   cmMendrelCathodeFrontAxisZ.commandConfiguration.camIn.deceleration := -1.0;
   cmMendrelCathodeFrontAxisZ.commandConfiguration.camIn.jerk := -1.0;
   cmMendrelCathodeFrontAxisZ.commandConfiguration.camIn.applicationMode := 0;
   cmMendrelCathodeFrontAxisZ.commandConfiguration.camIn.syncDirection := 1;
   cmMendrelCathodeFrontAxisZ.commandConfiguration.gearOutCamOut.slavePosition := 0.0;
   cmMendrelCathodeFrontAxisZ.commandConfiguration.gearOutCamOut.syncProfileReference := 1;
   cmMendrelCathodeFrontAxisZ.commandConfiguration.gearOutCamOut.masterStopDistance := 0.0;
   cmMendrelCathodeFrontAxisZ.commandConfiguration.gearOutCamOut.deceleration := -1.0;
   cmMendrelCathodeFrontAxisZ.commandConfiguration.gearOutCamOut.jerk := -1.0;
   cmMendrelCathodeFrontAxisZ.commandConfiguration.gearOutCamOut.syncOutDirection := 3;
   cmMendrelCathodeFrontAxisZ.commandConfiguration.gearOutCamOut.gearOutCamOutMode := -1;
   cmMendrelCathodeFrontAxisZ.commandConfiguration.phasing.phaseShift := 0.0;
   cmMendrelCathodeFrontAxisZ.commandConfiguration.phasing.velocity := -1.0;
   cmMendrelCathodeFrontAxisZ.commandConfiguration.phasing.acceleration := -1.0;
   cmMendrelCathodeFrontAxisZ.commandConfiguration.phasing.deceleration := -1.0;
   cmMendrelCathodeFrontAxisZ.commandConfiguration.phasing.jerk := -1.0;
   cmMendrelCathodeFrontAxisZ.commandConfiguration.phasing.profileReference := 0;
   cmMendrelCathodeFrontAxisZ.commandConfiguration.phasing.phasingDistance := 0.0;
   cmMendrelCathodeFrontAxisZ.commandConfiguration.phasing.startPosition := 0.0;
   cmMendrelCathodeFrontAxisZ.commandConfiguration.phasing.direction := 3;
   cmMendrelCathodeFrontAxisZ.commandConfiguration.phasing.phaseAbsolute := TRUE;
   cmMendrelCathodeFrontAxisZ.commandConfiguration.phasing.phaseShiftChangeOnTheFly := FALSE;
   cmMendrelCathodeFrontAxisZ.commandConfiguration.offset.offset := 0.0;
   cmMendrelCathodeFrontAxisZ.commandConfiguration.offset.profileReference := 1;
   cmMendrelCathodeFrontAxisZ.commandConfiguration.offset.offsetDistance := 0.0;
   cmMendrelCathodeFrontAxisZ.commandConfiguration.offset.startPosition := 0.0;
   cmMendrelCathodeFrontAxisZ.commandConfiguration.offset.direction := 3;
   cmMendrelCathodeFrontAxisZ.commandConfiguration.offset.offsetAbsolute := TRUE;
   cmMendrelCathodeFrontAxisZ.commandConfiguration.offset.offsetChangeOnTheFly := FALSE;
   cmMendrelCathodeFrontAxisZ.commands.enableMasterControl := TRUE;
   cmMendrelCathodeFrontAxisZ.commands.enableAxis := FALSE;
   cmMendrelCathodeFrontAxisZ.commands.resetAxis := FALSE;
   cmMendrelCathodeFrontAxisZ.commands.openBrake := FALSE;
   cmMendrelCathodeFrontAxisZ.commands.jogForward := FALSE;
   cmMendrelCathodeFrontAxisZ.commands.jogBackward := FALSE;
   cmMendrelCathodeFrontAxisZ.commands.moveVelocity := FALSE;
   cmMendrelCathodeFrontAxisZ.commands.stop := FALSE;
   cmMendrelCathodeFrontAxisZ.commands.fastStop := FALSE;
   cmMendrelCathodeFrontAxisZ.commands.torqueLimiting := FALSE;
   cmMendrelCathodeFrontAxisZ.commands.homing := FALSE;
   cmMendrelCathodeFrontAxisZ.commands.posRelative := FALSE;
   cmMendrelCathodeFrontAxisZ.commands.posAbsolute := FALSE;
   cmMendrelCathodeFrontAxisZ.commands.posSuperimposed := FALSE;
   cmMendrelCathodeFrontAxisZ.commands.haltSuperimposed := FALSE;
   cmMendrelCathodeFrontAxisZ.commands.selectSetPosition := 1;
   cmMendrelCathodeFrontAxisZ.commands.uploadParameters := FALSE;
   cmMendrelCathodeFrontAxisZ.commands.refreshConfiguration := FALSE;
   cmMendrelCathodeFrontAxisZ.commands.editConfiguration := FALSE;
   cmMendrelCathodeFrontAxisZ.commands.saveConfiguration := FALSE;
   cmMendrelCathodeFrontAxisZ.commands.uploadCurrentTorque := FALSE;
   cmMendrelCathodeFrontAxisZ.commands.reset := FALSE;
   cmMendrelCathodeFrontAxisZ.monitoring.enable := TRUE;
   cmMendrelCathodeFrontAxisZ.monitoring.referenceDesignator := WSTRING#'MendrelCathodeFrontAxisZ';
   cmMendrelCathodeFrontAxisZ.monitoring.enabled := TRUE;
   cmMendrelCathodeFrontAxisZ.monitoring.enableManualCmds := FALSE;
   cmMendrelCathodeFrontAxisZ.monitoring.reset := FALSE;
   cmMendrelCathodeFrontAxisZ.monitoring.resetAxis := FALSE;
   cmMendrelCathodeFrontAxisZ.monitoring.enableAxis := TRUE;
   cmMendrelCathodeFrontAxisZ.monitoring.openBrake := FALSE;
   cmMendrelCathodeFrontAxisZ.monitoring.jogBackward := FALSE;
   cmMendrelCathodeFrontAxisZ.monitoring.jogForward := FALSE;
   cmMendrelCathodeFrontAxisZ.monitoring.moveVelocity := FALSE;
   cmMendrelCathodeFrontAxisZ.monitoring.stop := FALSE;
   cmMendrelCathodeFrontAxisZ.monitoring.fastStop := FALSE;
   cmMendrelCathodeFrontAxisZ.monitoring.torqueLimiting := FALSE;
   cmMendrelCathodeFrontAxisZ.monitoring.homing := FALSE;
   cmMendrelCathodeFrontAxisZ.monitoring.posRelative := FALSE;
   cmMendrelCathodeFrontAxisZ.monitoring.posAbsolute := FALSE;
   cmMendrelCathodeFrontAxisZ.monitoring.posSuperimposed := FALSE;
   cmMendrelCathodeFrontAxisZ.monitoring.haltSuperimposed := FALSE;
   cmMendrelCathodeFrontAxisZ.monitoring.brakeOpened := FALSE;
   cmMendrelCathodeFrontAxisZ.monitoring.axisEnabled := TRUE;
   cmMendrelCathodeFrontAxisZ.monitoring.resetActive := FALSE;
   cmMendrelCathodeFrontAxisZ.monitoring.inVelocity := FALSE;
   cmMendrelCathodeFrontAxisZ.monitoring.inLimitation := FALSE;
   cmMendrelCathodeFrontAxisZ.monitoring.inClamping := FALSE;
   cmMendrelCathodeFrontAxisZ.monitoring.startSync := FALSE;
   cmMendrelCathodeFrontAxisZ.monitoring.inSync := FALSE;
   cmMendrelCathodeFrontAxisZ.monitoring.inSimulation := FALSE;
   cmMendrelCathodeFrontAxisZ.monitoring.jogSelected := FALSE;
   cmMendrelCathodeFrontAxisZ.monitoring.moveVelocitySelected := FALSE;
   cmMendrelCathodeFrontAxisZ.monitoring.stopSelected := FALSE;
   cmMendrelCathodeFrontAxisZ.monitoring.fastStopSelected := FALSE;
   cmMendrelCathodeFrontAxisZ.monitoring.torqueLimitingSelected := FALSE;
   cmMendrelCathodeFrontAxisZ.monitoring.homingSelected := FALSE;
   cmMendrelCathodeFrontAxisZ.monitoring.posRelativeSelected := FALSE;
   cmMendrelCathodeFrontAxisZ.monitoring.posAbsoluteSelected := FALSE;
   cmMendrelCathodeFrontAxisZ.monitoring.posSuperimposedSelected := FALSE;
   cmMendrelCathodeFrontAxisZ.monitoring.haltSuperimposedSelected := FALSE;
   cmMendrelCathodeFrontAxisZ.monitoring.commandBusy := FALSE;
   cmMendrelCathodeFrontAxisZ.monitoring.commandDone := FALSE;
   cmMendrelCathodeFrontAxisZ.monitoring.commandAborted := FALSE;
   cmMendrelCathodeFrontAxisZ.monitoring.homingCommandBusy := FALSE;
   cmMendrelCathodeFrontAxisZ.monitoring.homingCommandDone := FALSE;
   cmMendrelCathodeFrontAxisZ.monitoring.homingCommandAborted := FALSE;
   cmMendrelCathodeFrontAxisZ.monitoring.superimposedBusy := FALSE;
   cmMendrelCathodeFrontAxisZ.monitoring.superimposedDone := FALSE;
   cmMendrelCathodeFrontAxisZ.monitoring.superimposedAborted := FALSE;
   cmMendrelCathodeFrontAxisZ.monitoring.selectSetPosition := 1;
   cmMendrelCathodeFrontAxisZ.monitoring.selectionController := FALSE;
   cmMendrelCathodeFrontAxisZ.monitoring.interlockGeneral := TRUE;
   cmMendrelCathodeFrontAxisZ.monitoring.interlockJogForward := TRUE;
   cmMendrelCathodeFrontAxisZ.monitoring.interlockJogBackward := TRUE;
   cmMendrelCathodeFrontAxisZ.monitoring.interlockWarningGeneral := FALSE;
   cmMendrelCathodeFrontAxisZ.monitoring.interlockWarningJogForward := FALSE;
   cmMendrelCathodeFrontAxisZ.monitoring.interlockWarningJogBackward := FALSE;
   cmMendrelCathodeFrontAxisZ.monitoring.valid := TRUE;
   cmMendrelCathodeFrontAxisZ.monitoring.busy := TRUE;
   cmMendrelCathodeFrontAxisZ.monitoring.error := FALSE;
   cmMendrelCathodeFrontAxisZ.monitoring.status := 16#7002;
   cmMendrelCathodeFrontAxisZ.monitoring.subfunctionStatus := 16#0000;
   cmMendrelCathodeFrontAxisZ.monitoring.actualPosition := 50.0;
   cmMendrelCathodeFrontAxisZ.monitoring.actualSpeed := 0.0;
   cmMendrelCathodeFrontAxisZ.monitoring.speedUnit := 1062;
   cmMendrelCathodeFrontAxisZ.monitoring.positionUnit := 1013;
   cmMendrelCathodeFrontAxisZ.monitoring.axisStatus1 := 16#0240_10A1;
   cmMendrelCathodeFrontAxisZ.monitoring.axisStatus2 := 16#0000_0000;
   cmMendrelCathodeFrontAxisZ.monitoring.axisType := 1;
   cmMendrelCathodeFrontAxisZ.monitoring.maxVelocity := 2500.0;
   cmMendrelCathodeFrontAxisZ.monitoring.actualCurrent := 0.0;
   cmMendrelCathodeFrontAxisZ.monitoring.actualTorque := 0.0;
   cmMendrelCathodeFrontAxisZ.monitoring.velocityOverrideEnabled := FALSE;
   cmMendrelCathodeFrontAxisZ.monitoring.sinaParaError := FALSE;
   cmMendrelCathodeFrontAxisZ.monitoring.sinaParaStatus := 16#0000_0000;
   cmMendrelCathodeFrontAxisZ.configuration.referenceDesignator := WSTRING#'MendrelCathodeFrontAxisZ';
   cmMendrelCathodeFrontAxisZ.configuration.disableAlarms := FALSE;
   cmMendrelCathodeFrontAxisZ.configuration.masterControlPopUp := TRUE;
   cmMendrelCathodeFrontAxisZ.configuration.setPositions[0].position := 0.0;
   cmMendrelCathodeFrontAxisZ.configuration.setPositions[1].position := 50.0;
   cmMendrelCathodeFrontAxisZ.configuration.setPositions[2..15].position := 0.0;
   cmMendrelCathodeFrontAxisZ.configuration.setPositions[0..1].velocity := 50.0;
   cmMendrelCathodeFrontAxisZ.configuration.setPositions[2..15].velocity := -1.0;
   cmMendrelCathodeFrontAxisZ.configuration.setPositions[0..1].acceleration := 500.0;
   cmMendrelCathodeFrontAxisZ.configuration.setPositions[2..15].acceleration := -1.0;
   cmMendrelCathodeFrontAxisZ.configuration.setPositions[0..1].deceleration := 500.0;
   cmMendrelCathodeFrontAxisZ.configuration.setPositions[2..15].deceleration := -1.0;
   cmMendrelCathodeFrontAxisZ.configuration.setPositions[0..15]."name" := '';
   cmMendrelCathodeRearAxisY.commandConfiguration.generalSettings.stopOnError := TRUE;
   cmMendrelCathodeRearAxisY.commandConfiguration.generalSettings.resetWithRestart := FALSE;
   cmMendrelCathodeRearAxisY.commandConfiguration.generalSettings.abortWaitingSyncCmd := TRUE;
   cmMendrelCathodeRearAxisY.commandConfiguration.power.startMode := 1;
   cmMendrelCathodeRearAxisY.commandConfiguration.power.stopMode := 0;
   cmMendrelCathodeRearAxisY.commandConfiguration.power.syncMotionSimulation := FALSE;
   cmMendrelCathodeRearAxisY.commandConfiguration.power.syncMotionSimulationExtendedMode := -1;
   cmMendrelCathodeRearAxisY.commandConfiguration.jog.velocity := 0.0;
   cmMendrelCathodeRearAxisY.commandConfiguration.jog.acceleration := -1.0;
   cmMendrelCathodeRearAxisY.commandConfiguration.jog.deceleration := -1.0;
   cmMendrelCathodeRearAxisY.commandConfiguration.jog.jerk := -1.0;
   cmMendrelCathodeRearAxisY.commandConfiguration.jog.positionControlled := TRUE;
   cmMendrelCathodeRearAxisY.commandConfiguration.jog.increment := 0.0;
   cmMendrelCathodeRearAxisY.commandConfiguration.jog.mode := 0;
   cmMendrelCathodeRearAxisY.commandConfiguration.moveVelocity.velocity := 0.0;
   cmMendrelCathodeRearAxisY.commandConfiguration.moveVelocity.acceleration := -1.0;
   cmMendrelCathodeRearAxisY.commandConfiguration.moveVelocity.deceleration := -1.0;
   cmMendrelCathodeRearAxisY.commandConfiguration.moveVelocity.jerk := -1.0;
   cmMendrelCathodeRearAxisY.commandConfiguration.moveVelocity.direction := 0;
   cmMendrelCathodeRearAxisY.commandConfiguration.moveVelocity.positionControlled := TRUE;
   cmMendrelCathodeRearAxisY.commandConfiguration.moveVelocity.velocityChangeOnTheFly := FALSE;
   cmMendrelCathodeRearAxisY.commandConfiguration.stop.deceleration := -1.0;
   cmMendrelCathodeRearAxisY.commandConfiguration.stop.jerk := -1.0;
   cmMendrelCathodeRearAxisY.commandConfiguration.stop.abortAcceleration := FALSE;
   cmMendrelCathodeRearAxisY.commandConfiguration.fastStop.deceleration := -1.0;
   cmMendrelCathodeRearAxisY.commandConfiguration.fastStop.jerk := -1.0;
   cmMendrelCathodeRearAxisY.commandConfiguration.fastStop.abortAcceleration := FALSE;
   cmMendrelCathodeRearAxisY.commandConfiguration.fastStop.replaceStopPossible := FALSE;
   cmMendrelCathodeRearAxisY.commandConfiguration.torqueLimiting.limit := -1.0;
   cmMendrelCathodeRearAxisY.commandConfiguration.torqueLimiting.mode := 0;
   cmMendrelCathodeRearAxisY.commandConfiguration.homing.position := 0.0;
   cmMendrelCathodeRearAxisY.commandConfiguration.homing.mode := 0;
   cmMendrelCathodeRearAxisY.commandConfiguration.homing.sensor := 0;
   cmMendrelCathodeRearAxisY.commandConfiguration.homing.extendedMode := -1;
   cmMendrelCathodeRearAxisY.commandConfiguration.homing.extendedModeTorqueLimit := 0.0;
   cmMendrelCathodeRearAxisY.commandConfiguration.homing.extendedModeTargetPosition := 0.0;
   cmMendrelCathodeRearAxisY.commandConfiguration.posRelative.distance := 0.0;
   cmMendrelCathodeRearAxisY.commandConfiguration.posRelative.velocity := -1.0;
   cmMendrelCathodeRearAxisY.commandConfiguration.posRelative.acceleration := -1.0;
   cmMendrelCathodeRearAxisY.commandConfiguration.posRelative.deceleration := -1.0;
   cmMendrelCathodeRearAxisY.commandConfiguration.posRelative.jerk := -1.0;
   cmMendrelCathodeRearAxisY.commandConfiguration.posRelative.direction := 0;
   cmMendrelCathodeRearAxisY.commandConfiguration.posAbsolute.position := 0.0;
   cmMendrelCathodeRearAxisY.commandConfiguration.posAbsolute.velocity := -1.0;
   cmMendrelCathodeRearAxisY.commandConfiguration.posAbsolute.acceleration := -1.0;
   cmMendrelCathodeRearAxisY.commandConfiguration.posAbsolute.deceleration := -1.0;
   cmMendrelCathodeRearAxisY.commandConfiguration.posAbsolute.jerk := -1.0;
   cmMendrelCathodeRearAxisY.commandConfiguration.posAbsolute.direction := 1;
   cmMendrelCathodeRearAxisY.commandConfiguration.posAbsolute.positionChangeOnTheFly := FALSE;
   cmMendrelCathodeRearAxisY.commandConfiguration.posAbsolute.velocityChangeOnTheFly := FALSE;
   cmMendrelCathodeRearAxisY.commandConfiguration.posSuperimposed.distance := 0.0;
   cmMendrelCathodeRearAxisY.commandConfiguration.posSuperimposed.velocityDiff := -1.0;
   cmMendrelCathodeRearAxisY.commandConfiguration.posSuperimposed.acceleration := -1.0;
   cmMendrelCathodeRearAxisY.commandConfiguration.posSuperimposed.deceleration := -1.0;
   cmMendrelCathodeRearAxisY.commandConfiguration.posSuperimposed.jerk := -1.0;
   cmMendrelCathodeRearAxisY.commandConfiguration.posSuperimposed.direction := 0;
   cmMendrelCathodeRearAxisY.commandConfiguration.haltSuperimposed.deceleration := -1.0;
   cmMendrelCathodeRearAxisY.commandConfiguration.haltSuperimposed.jerk := -1.0;
   cmMendrelCathodeRearAxisY.commandConfiguration.haltSuperimposed.abortAcceleration := FALSE;
   cmMendrelCathodeRearAxisY.commandConfiguration.gearInRelative.ratioNumerator := 1;
   cmMendrelCathodeRearAxisY.commandConfiguration.gearInRelative.ratioDenominator := 1;
   cmMendrelCathodeRearAxisY.commandConfiguration.gearInRelative.acceleration := -1.0;
   cmMendrelCathodeRearAxisY.commandConfiguration.gearInRelative.deceleration := -1.0;
   cmMendrelCathodeRearAxisY.commandConfiguration.gearInRelative.jerk := -1.0;
   cmMendrelCathodeRearAxisY.commandConfiguration.gearInRelative.ratioChangeOnTheFly := FALSE;
   cmMendrelCathodeRearAxisY.commandConfiguration.gearInAbsolute.ratioNumerator := 1;
   cmMendrelCathodeRearAxisY.commandConfiguration.gearInAbsolute.ratioDenominator := 1;
   cmMendrelCathodeRearAxisY.commandConfiguration.gearInAbsolute.masterSyncPosition := 0.0;
   cmMendrelCathodeRearAxisY.commandConfiguration.gearInAbsolute.slaveSyncPosition := 0.0;
   cmMendrelCathodeRearAxisY.commandConfiguration.gearInAbsolute.syncProfileReference := 1;
   cmMendrelCathodeRearAxisY.commandConfiguration.gearInAbsolute.masterStartDistance := 0.0;
   cmMendrelCathodeRearAxisY.commandConfiguration.gearInAbsolute.velocity := -1.0;
   cmMendrelCathodeRearAxisY.commandConfiguration.gearInAbsolute.acceleration := -1.0;
   cmMendrelCathodeRearAxisY.commandConfiguration.gearInAbsolute.deceleration := -1.0;
   cmMendrelCathodeRearAxisY.commandConfiguration.gearInAbsolute.jerk := -1.0;
   cmMendrelCathodeRearAxisY.commandConfiguration.gearInAbsolute.syncDirection := 1;
   cmMendrelCathodeRearAxisY.commandConfiguration.gearInAbsolute.ratioChangeOnTheFly := FALSE;
   cmMendrelCathodeRearAxisY.commandConfiguration.gearInVelocity.continuousUpdate := FALSE;
   cmMendrelCathodeRearAxisY.commandConfiguration.gearInVelocity.ratioNumerator := 1;
   cmMendrelCathodeRearAxisY.commandConfiguration.gearInVelocity.ratioDenominator := 1;
   cmMendrelCathodeRearAxisY.commandConfiguration.gearInVelocity.acceleration := -1.0;
   cmMendrelCathodeRearAxisY.commandConfiguration.gearInVelocity.deceleration := -1.0;
   cmMendrelCathodeRearAxisY.commandConfiguration.gearInVelocity.jerk := -1.0;
   cmMendrelCathodeRearAxisY.commandConfiguration.gearInVelocity.positionControlled := FALSE;
   cmMendrelCathodeRearAxisY.commandConfiguration.camIn.masterOffset := 0.0;
   cmMendrelCathodeRearAxisY.commandConfiguration.camIn.slaveOffset := 0.0;
   cmMendrelCathodeRearAxisY.commandConfiguration.camIn.masterScaling := 1.0;
   cmMendrelCathodeRearAxisY.commandConfiguration.camIn.slaveScaling := 1.0;
   cmMendrelCathodeRearAxisY.commandConfiguration.camIn.masterSyncPosition := 0.0;
   cmMendrelCathodeRearAxisY.commandConfiguration.camIn.syncProfileReference := 1;
   cmMendrelCathodeRearAxisY.commandConfiguration.camIn.masterStartDistance := 0.0;
   cmMendrelCathodeRearAxisY.commandConfiguration.camIn.velocity := -1.0;
   cmMendrelCathodeRearAxisY.commandConfiguration.camIn.acceleration := -1.0;
   cmMendrelCathodeRearAxisY.commandConfiguration.camIn.deceleration := -1.0;
   cmMendrelCathodeRearAxisY.commandConfiguration.camIn.jerk := -1.0;
   cmMendrelCathodeRearAxisY.commandConfiguration.camIn.applicationMode := 0;
   cmMendrelCathodeRearAxisY.commandConfiguration.camIn.syncDirection := 1;
   cmMendrelCathodeRearAxisY.commandConfiguration.gearOutCamOut.slavePosition := 0.0;
   cmMendrelCathodeRearAxisY.commandConfiguration.gearOutCamOut.syncProfileReference := 1;
   cmMendrelCathodeRearAxisY.commandConfiguration.gearOutCamOut.masterStopDistance := 0.0;
   cmMendrelCathodeRearAxisY.commandConfiguration.gearOutCamOut.deceleration := -1.0;
   cmMendrelCathodeRearAxisY.commandConfiguration.gearOutCamOut.jerk := -1.0;
   cmMendrelCathodeRearAxisY.commandConfiguration.gearOutCamOut.syncOutDirection := 3;
   cmMendrelCathodeRearAxisY.commandConfiguration.gearOutCamOut.gearOutCamOutMode := -1;
   cmMendrelCathodeRearAxisY.commandConfiguration.phasing.phaseShift := 0.0;
   cmMendrelCathodeRearAxisY.commandConfiguration.phasing.velocity := -1.0;
   cmMendrelCathodeRearAxisY.commandConfiguration.phasing.acceleration := -1.0;
   cmMendrelCathodeRearAxisY.commandConfiguration.phasing.deceleration := -1.0;
   cmMendrelCathodeRearAxisY.commandConfiguration.phasing.jerk := -1.0;
   cmMendrelCathodeRearAxisY.commandConfiguration.phasing.profileReference := 0;
   cmMendrelCathodeRearAxisY.commandConfiguration.phasing.phasingDistance := 0.0;
   cmMendrelCathodeRearAxisY.commandConfiguration.phasing.startPosition := 0.0;
   cmMendrelCathodeRearAxisY.commandConfiguration.phasing.direction := 3;
   cmMendrelCathodeRearAxisY.commandConfiguration.phasing.phaseAbsolute := TRUE;
   cmMendrelCathodeRearAxisY.commandConfiguration.phasing.phaseShiftChangeOnTheFly := FALSE;
   cmMendrelCathodeRearAxisY.commandConfiguration.offset.offset := 0.0;
   cmMendrelCathodeRearAxisY.commandConfiguration.offset.profileReference := 1;
   cmMendrelCathodeRearAxisY.commandConfiguration.offset.offsetDistance := 0.0;
   cmMendrelCathodeRearAxisY.commandConfiguration.offset.startPosition := 0.0;
   cmMendrelCathodeRearAxisY.commandConfiguration.offset.direction := 3;
   cmMendrelCathodeRearAxisY.commandConfiguration.offset.offsetAbsolute := TRUE;
   cmMendrelCathodeRearAxisY.commandConfiguration.offset.offsetChangeOnTheFly := FALSE;
   cmMendrelCathodeRearAxisY.commands.enableMasterControl := TRUE;
   cmMendrelCathodeRearAxisY.commands.enableAxis := FALSE;
   cmMendrelCathodeRearAxisY.commands.resetAxis := FALSE;
   cmMendrelCathodeRearAxisY.commands.openBrake := FALSE;
   cmMendrelCathodeRearAxisY.commands.jogForward := FALSE;
   cmMendrelCathodeRearAxisY.commands.jogBackward := FALSE;
   cmMendrelCathodeRearAxisY.commands.moveVelocity := FALSE;
   cmMendrelCathodeRearAxisY.commands.stop := FALSE;
   cmMendrelCathodeRearAxisY.commands.fastStop := FALSE;
   cmMendrelCathodeRearAxisY.commands.torqueLimiting := FALSE;
   cmMendrelCathodeRearAxisY.commands.homing := FALSE;
   cmMendrelCathodeRearAxisY.commands.posRelative := FALSE;
   cmMendrelCathodeRearAxisY.commands.posAbsolute := FALSE;
   cmMendrelCathodeRearAxisY.commands.posSuperimposed := FALSE;
   cmMendrelCathodeRearAxisY.commands.haltSuperimposed := FALSE;
   cmMendrelCathodeRearAxisY.commands.selectSetPosition := 1;
   cmMendrelCathodeRearAxisY.commands.uploadParameters := FALSE;
   cmMendrelCathodeRearAxisY.commands.refreshConfiguration := FALSE;
   cmMendrelCathodeRearAxisY.commands.editConfiguration := FALSE;
   cmMendrelCathodeRearAxisY.commands.saveConfiguration := FALSE;
   cmMendrelCathodeRearAxisY.commands.uploadCurrentTorque := FALSE;
   cmMendrelCathodeRearAxisY.commands.reset := FALSE;
   cmMendrelCathodeRearAxisY.monitoring.enable := TRUE;
   cmMendrelCathodeRearAxisY.monitoring.referenceDesignator := WSTRING#'MendrelCathodeRearAxisY';
   cmMendrelCathodeRearAxisY.monitoring.enabled := TRUE;
   cmMendrelCathodeRearAxisY.monitoring.enableManualCmds := FALSE;
   cmMendrelCathodeRearAxisY.monitoring.reset := FALSE;
   cmMendrelCathodeRearAxisY.monitoring.resetAxis := FALSE;
   cmMendrelCathodeRearAxisY.monitoring.enableAxis := TRUE;
   cmMendrelCathodeRearAxisY.monitoring.openBrake := FALSE;
   cmMendrelCathodeRearAxisY.monitoring.jogBackward := FALSE;
   cmMendrelCathodeRearAxisY.monitoring.jogForward := FALSE;
   cmMendrelCathodeRearAxisY.monitoring.moveVelocity := FALSE;
   cmMendrelCathodeRearAxisY.monitoring.stop := FALSE;
   cmMendrelCathodeRearAxisY.monitoring.fastStop := FALSE;
   cmMendrelCathodeRearAxisY.monitoring.torqueLimiting := FALSE;
   cmMendrelCathodeRearAxisY.monitoring.homing := FALSE;
   cmMendrelCathodeRearAxisY.monitoring.posRelative := FALSE;
   cmMendrelCathodeRearAxisY.monitoring.posAbsolute := FALSE;
   cmMendrelCathodeRearAxisY.monitoring.posSuperimposed := FALSE;
   cmMendrelCathodeRearAxisY.monitoring.haltSuperimposed := FALSE;
   cmMendrelCathodeRearAxisY.monitoring.brakeOpened := FALSE;
   cmMendrelCathodeRearAxisY.monitoring.axisEnabled := TRUE;
   cmMendrelCathodeRearAxisY.monitoring.resetActive := FALSE;
   cmMendrelCathodeRearAxisY.monitoring.inVelocity := FALSE;
   cmMendrelCathodeRearAxisY.monitoring.inLimitation := FALSE;
   cmMendrelCathodeRearAxisY.monitoring.inClamping := FALSE;
   cmMendrelCathodeRearAxisY.monitoring.startSync := FALSE;
   cmMendrelCathodeRearAxisY.monitoring.inSync := FALSE;
   cmMendrelCathodeRearAxisY.monitoring.inSimulation := FALSE;
   cmMendrelCathodeRearAxisY.monitoring.jogSelected := FALSE;
   cmMendrelCathodeRearAxisY.monitoring.moveVelocitySelected := FALSE;
   cmMendrelCathodeRearAxisY.monitoring.stopSelected := FALSE;
   cmMendrelCathodeRearAxisY.monitoring.fastStopSelected := FALSE;
   cmMendrelCathodeRearAxisY.monitoring.torqueLimitingSelected := FALSE;
   cmMendrelCathodeRearAxisY.monitoring.homingSelected := FALSE;
   cmMendrelCathodeRearAxisY.monitoring.posRelativeSelected := FALSE;
   cmMendrelCathodeRearAxisY.monitoring.posAbsoluteSelected := FALSE;
   cmMendrelCathodeRearAxisY.monitoring.posSuperimposedSelected := FALSE;
   cmMendrelCathodeRearAxisY.monitoring.haltSuperimposedSelected := FALSE;
   cmMendrelCathodeRearAxisY.monitoring.commandBusy := FALSE;
   cmMendrelCathodeRearAxisY.monitoring.commandDone := FALSE;
   cmMendrelCathodeRearAxisY.monitoring.commandAborted := FALSE;
   cmMendrelCathodeRearAxisY.monitoring.homingCommandBusy := FALSE;
   cmMendrelCathodeRearAxisY.monitoring.homingCommandDone := FALSE;
   cmMendrelCathodeRearAxisY.monitoring.homingCommandAborted := FALSE;
   cmMendrelCathodeRearAxisY.monitoring.superimposedBusy := FALSE;
   cmMendrelCathodeRearAxisY.monitoring.superimposedDone := FALSE;
   cmMendrelCathodeRearAxisY.monitoring.superimposedAborted := FALSE;
   cmMendrelCathodeRearAxisY.monitoring.selectSetPosition := 1;
   cmMendrelCathodeRearAxisY.monitoring.selectionController := FALSE;
   cmMendrelCathodeRearAxisY.monitoring.interlockGeneral := TRUE;
   cmMendrelCathodeRearAxisY.monitoring.interlockJogForward := TRUE;
   cmMendrelCathodeRearAxisY.monitoring.interlockJogBackward := TRUE;
   cmMendrelCathodeRearAxisY.monitoring.interlockWarningGeneral := FALSE;
   cmMendrelCathodeRearAxisY.monitoring.interlockWarningJogForward := FALSE;
   cmMendrelCathodeRearAxisY.monitoring.interlockWarningJogBackward := FALSE;
   cmMendrelCathodeRearAxisY.monitoring.valid := TRUE;
   cmMendrelCathodeRearAxisY.monitoring.busy := TRUE;
   cmMendrelCathodeRearAxisY.monitoring.error := FALSE;
   cmMendrelCathodeRearAxisY.monitoring.status := 16#7002;
   cmMendrelCathodeRearAxisY.monitoring.subfunctionStatus := 16#0000;
   cmMendrelCathodeRearAxisY.monitoring.actualPosition := 0.0;
   cmMendrelCathodeRearAxisY.monitoring.actualSpeed := 0.0;
   cmMendrelCathodeRearAxisY.monitoring.speedUnit := 1062;
   cmMendrelCathodeRearAxisY.monitoring.positionUnit := 1013;
   cmMendrelCathodeRearAxisY.monitoring.axisStatus1 := 16#0240_10A1;
   cmMendrelCathodeRearAxisY.monitoring.axisStatus2 := 16#0000_0000;
   cmMendrelCathodeRearAxisY.monitoring.axisType := 1;
   cmMendrelCathodeRearAxisY.monitoring.maxVelocity := 2500.0;
   cmMendrelCathodeRearAxisY.monitoring.actualCurrent := 0.0;
   cmMendrelCathodeRearAxisY.monitoring.actualTorque := 0.0;
   cmMendrelCathodeRearAxisY.monitoring.velocityOverrideEnabled := FALSE;
   cmMendrelCathodeRearAxisY.monitoring.sinaParaError := FALSE;
   cmMendrelCathodeRearAxisY.monitoring.sinaParaStatus := 16#0000_0000;
   cmMendrelCathodeRearAxisY.configuration.referenceDesignator := WSTRING#'MendrelCathodeRearAxisY';
   cmMendrelCathodeRearAxisY.configuration.disableAlarms := FALSE;
   cmMendrelCathodeRearAxisY.configuration.masterControlPopUp := TRUE;
   cmMendrelCathodeRearAxisY.configuration.setPositions[0].position := 0.0;
   cmMendrelCathodeRearAxisY.configuration.setPositions[1].position := 50.0;
   cmMendrelCathodeRearAxisY.configuration.setPositions[2..15].position := 0.0;
   cmMendrelCathodeRearAxisY.configuration.setPositions[0..1].velocity := 50.0;
   cmMendrelCathodeRearAxisY.configuration.setPositions[2..15].velocity := -1.0;
   cmMendrelCathodeRearAxisY.configuration.setPositions[0..1].acceleration := 500.0;
   cmMendrelCathodeRearAxisY.configuration.setPositions[2..15].acceleration := -1.0;
   cmMendrelCathodeRearAxisY.configuration.setPositions[0..1].deceleration := 500.0;
   cmMendrelCathodeRearAxisY.configuration.setPositions[2..15].deceleration := -1.0;
   cmMendrelCathodeRearAxisY.configuration.setPositions[0..15]."name" := '';
   cmMendrelCathodeRearAxisZ.commandConfiguration.generalSettings.stopOnError := TRUE;
   cmMendrelCathodeRearAxisZ.commandConfiguration.generalSettings.resetWithRestart := FALSE;
   cmMendrelCathodeRearAxisZ.commandConfiguration.generalSettings.abortWaitingSyncCmd := TRUE;
   cmMendrelCathodeRearAxisZ.commandConfiguration.power.startMode := 1;
   cmMendrelCathodeRearAxisZ.commandConfiguration.power.stopMode := 0;
   cmMendrelCathodeRearAxisZ.commandConfiguration.power.syncMotionSimulation := FALSE;
   cmMendrelCathodeRearAxisZ.commandConfiguration.power.syncMotionSimulationExtendedMode := -1;
   cmMendrelCathodeRearAxisZ.commandConfiguration.jog.velocity := 0.0;
   cmMendrelCathodeRearAxisZ.commandConfiguration.jog.acceleration := -1.0;
   cmMendrelCathodeRearAxisZ.commandConfiguration.jog.deceleration := -1.0;
   cmMendrelCathodeRearAxisZ.commandConfiguration.jog.jerk := -1.0;
   cmMendrelCathodeRearAxisZ.commandConfiguration.jog.positionControlled := TRUE;
   cmMendrelCathodeRearAxisZ.commandConfiguration.jog.increment := 0.0;
   cmMendrelCathodeRearAxisZ.commandConfiguration.jog.mode := 0;
   cmMendrelCathodeRearAxisZ.commandConfiguration.moveVelocity.velocity := 0.0;
   cmMendrelCathodeRearAxisZ.commandConfiguration.moveVelocity.acceleration := -1.0;
   cmMendrelCathodeRearAxisZ.commandConfiguration.moveVelocity.deceleration := -1.0;
   cmMendrelCathodeRearAxisZ.commandConfiguration.moveVelocity.jerk := -1.0;
   cmMendrelCathodeRearAxisZ.commandConfiguration.moveVelocity.direction := 0;
   cmMendrelCathodeRearAxisZ.commandConfiguration.moveVelocity.positionControlled := TRUE;
   cmMendrelCathodeRearAxisZ.commandConfiguration.moveVelocity.velocityChangeOnTheFly := FALSE;
   cmMendrelCathodeRearAxisZ.commandConfiguration.stop.deceleration := -1.0;
   cmMendrelCathodeRearAxisZ.commandConfiguration.stop.jerk := -1.0;
   cmMendrelCathodeRearAxisZ.commandConfiguration.stop.abortAcceleration := FALSE;
   cmMendrelCathodeRearAxisZ.commandConfiguration.fastStop.deceleration := -1.0;
   cmMendrelCathodeRearAxisZ.commandConfiguration.fastStop.jerk := -1.0;
   cmMendrelCathodeRearAxisZ.commandConfiguration.fastStop.abortAcceleration := FALSE;
   cmMendrelCathodeRearAxisZ.commandConfiguration.fastStop.replaceStopPossible := FALSE;
   cmMendrelCathodeRearAxisZ.commandConfiguration.torqueLimiting.limit := -1.0;
   cmMendrelCathodeRearAxisZ.commandConfiguration.torqueLimiting.mode := 0;
   cmMendrelCathodeRearAxisZ.commandConfiguration.homing.position := 0.0;
   cmMendrelCathodeRearAxisZ.commandConfiguration.homing.mode := 0;
   cmMendrelCathodeRearAxisZ.commandConfiguration.homing.sensor := 0;
   cmMendrelCathodeRearAxisZ.commandConfiguration.homing.extendedMode := -1;
   cmMendrelCathodeRearAxisZ.commandConfiguration.homing.extendedModeTorqueLimit := 0.0;
   cmMendrelCathodeRearAxisZ.commandConfiguration.homing.extendedModeTargetPosition := 0.0;
   cmMendrelCathodeRearAxisZ.commandConfiguration.posRelative.distance := 0.0;
   cmMendrelCathodeRearAxisZ.commandConfiguration.posRelative.velocity := -1.0;
   cmMendrelCathodeRearAxisZ.commandConfiguration.posRelative.acceleration := -1.0;
   cmMendrelCathodeRearAxisZ.commandConfiguration.posRelative.deceleration := -1.0;
   cmMendrelCathodeRearAxisZ.commandConfiguration.posRelative.jerk := -1.0;
   cmMendrelCathodeRearAxisZ.commandConfiguration.posRelative.direction := 0;
   cmMendrelCathodeRearAxisZ.commandConfiguration.posAbsolute.position := 0.0;
   cmMendrelCathodeRearAxisZ.commandConfiguration.posAbsolute.velocity := -1.0;
   cmMendrelCathodeRearAxisZ.commandConfiguration.posAbsolute.acceleration := -1.0;
   cmMendrelCathodeRearAxisZ.commandConfiguration.posAbsolute.deceleration := -1.0;
   cmMendrelCathodeRearAxisZ.commandConfiguration.posAbsolute.jerk := -1.0;
   cmMendrelCathodeRearAxisZ.commandConfiguration.posAbsolute.direction := 1;
   cmMendrelCathodeRearAxisZ.commandConfiguration.posAbsolute.positionChangeOnTheFly := FALSE;
   cmMendrelCathodeRearAxisZ.commandConfiguration.posAbsolute.velocityChangeOnTheFly := FALSE;
   cmMendrelCathodeRearAxisZ.commandConfiguration.posSuperimposed.distance := 0.0;
   cmMendrelCathodeRearAxisZ.commandConfiguration.posSuperimposed.velocityDiff := -1.0;
   cmMendrelCathodeRearAxisZ.commandConfiguration.posSuperimposed.acceleration := -1.0;
   cmMendrelCathodeRearAxisZ.commandConfiguration.posSuperimposed.deceleration := -1.0;
   cmMendrelCathodeRearAxisZ.commandConfiguration.posSuperimposed.jerk := -1.0;
   cmMendrelCathodeRearAxisZ.commandConfiguration.posSuperimposed.direction := 0;
   cmMendrelCathodeRearAxisZ.commandConfiguration.haltSuperimposed.deceleration := -1.0;
   cmMendrelCathodeRearAxisZ.commandConfiguration.haltSuperimposed.jerk := -1.0;
   cmMendrelCathodeRearAxisZ.commandConfiguration.haltSuperimposed.abortAcceleration := FALSE;
   cmMendrelCathodeRearAxisZ.commandConfiguration.gearInRelative.ratioNumerator := 1;
   cmMendrelCathodeRearAxisZ.commandConfiguration.gearInRelative.ratioDenominator := 1;
   cmMendrelCathodeRearAxisZ.commandConfiguration.gearInRelative.acceleration := -1.0;
   cmMendrelCathodeRearAxisZ.commandConfiguration.gearInRelative.deceleration := -1.0;
   cmMendrelCathodeRearAxisZ.commandConfiguration.gearInRelative.jerk := -1.0;
   cmMendrelCathodeRearAxisZ.commandConfiguration.gearInRelative.ratioChangeOnTheFly := FALSE;
   cmMendrelCathodeRearAxisZ.commandConfiguration.gearInAbsolute.ratioNumerator := 1;
   cmMendrelCathodeRearAxisZ.commandConfiguration.gearInAbsolute.ratioDenominator := 1;
   cmMendrelCathodeRearAxisZ.commandConfiguration.gearInAbsolute.masterSyncPosition := 0.0;
   cmMendrelCathodeRearAxisZ.commandConfiguration.gearInAbsolute.slaveSyncPosition := 0.0;
   cmMendrelCathodeRearAxisZ.commandConfiguration.gearInAbsolute.syncProfileReference := 1;
   cmMendrelCathodeRearAxisZ.commandConfiguration.gearInAbsolute.masterStartDistance := 0.0;
   cmMendrelCathodeRearAxisZ.commandConfiguration.gearInAbsolute.velocity := -1.0;
   cmMendrelCathodeRearAxisZ.commandConfiguration.gearInAbsolute.acceleration := -1.0;
   cmMendrelCathodeRearAxisZ.commandConfiguration.gearInAbsolute.deceleration := -1.0;
   cmMendrelCathodeRearAxisZ.commandConfiguration.gearInAbsolute.jerk := -1.0;
   cmMendrelCathodeRearAxisZ.commandConfiguration.gearInAbsolute.syncDirection := 1;
   cmMendrelCathodeRearAxisZ.commandConfiguration.gearInAbsolute.ratioChangeOnTheFly := FALSE;
   cmMendrelCathodeRearAxisZ.commandConfiguration.gearInVelocity.continuousUpdate := FALSE;
   cmMendrelCathodeRearAxisZ.commandConfiguration.gearInVelocity.ratioNumerator := 1;
   cmMendrelCathodeRearAxisZ.commandConfiguration.gearInVelocity.ratioDenominator := 1;
   cmMendrelCathodeRearAxisZ.commandConfiguration.gearInVelocity.acceleration := -1.0;
   cmMendrelCathodeRearAxisZ.commandConfiguration.gearInVelocity.deceleration := -1.0;
   cmMendrelCathodeRearAxisZ.commandConfiguration.gearInVelocity.jerk := -1.0;
   cmMendrelCathodeRearAxisZ.commandConfiguration.gearInVelocity.positionControlled := FALSE;
   cmMendrelCathodeRearAxisZ.commandConfiguration.camIn.masterOffset := 0.0;
   cmMendrelCathodeRearAxisZ.commandConfiguration.camIn.slaveOffset := 0.0;
   cmMendrelCathodeRearAxisZ.commandConfiguration.camIn.masterScaling := 1.0;
   cmMendrelCathodeRearAxisZ.commandConfiguration.camIn.slaveScaling := 1.0;
   cmMendrelCathodeRearAxisZ.commandConfiguration.camIn.masterSyncPosition := 0.0;
   cmMendrelCathodeRearAxisZ.commandConfiguration.camIn.syncProfileReference := 1;
   cmMendrelCathodeRearAxisZ.commandConfiguration.camIn.masterStartDistance := 0.0;
   cmMendrelCathodeRearAxisZ.commandConfiguration.camIn.velocity := -1.0;
   cmMendrelCathodeRearAxisZ.commandConfiguration.camIn.acceleration := -1.0;
   cmMendrelCathodeRearAxisZ.commandConfiguration.camIn.deceleration := -1.0;
   cmMendrelCathodeRearAxisZ.commandConfiguration.camIn.jerk := -1.0;
   cmMendrelCathodeRearAxisZ.commandConfiguration.camIn.applicationMode := 0;
   cmMendrelCathodeRearAxisZ.commandConfiguration.camIn.syncDirection := 1;
   cmMendrelCathodeRearAxisZ.commandConfiguration.gearOutCamOut.slavePosition := 0.0;
   cmMendrelCathodeRearAxisZ.commandConfiguration.gearOutCamOut.syncProfileReference := 1;
   cmMendrelCathodeRearAxisZ.commandConfiguration.gearOutCamOut.masterStopDistance := 0.0;
   cmMendrelCathodeRearAxisZ.commandConfiguration.gearOutCamOut.deceleration := -1.0;
   cmMendrelCathodeRearAxisZ.commandConfiguration.gearOutCamOut.jerk := -1.0;
   cmMendrelCathodeRearAxisZ.commandConfiguration.gearOutCamOut.syncOutDirection := 3;
   cmMendrelCathodeRearAxisZ.commandConfiguration.gearOutCamOut.gearOutCamOutMode := -1;
   cmMendrelCathodeRearAxisZ.commandConfiguration.phasing.phaseShift := 0.0;
   cmMendrelCathodeRearAxisZ.commandConfiguration.phasing.velocity := -1.0;
   cmMendrelCathodeRearAxisZ.commandConfiguration.phasing.acceleration := -1.0;
   cmMendrelCathodeRearAxisZ.commandConfiguration.phasing.deceleration := -1.0;
   cmMendrelCathodeRearAxisZ.commandConfiguration.phasing.jerk := -1.0;
   cmMendrelCathodeRearAxisZ.commandConfiguration.phasing.profileReference := 0;
   cmMendrelCathodeRearAxisZ.commandConfiguration.phasing.phasingDistance := 0.0;
   cmMendrelCathodeRearAxisZ.commandConfiguration.phasing.startPosition := 0.0;
   cmMendrelCathodeRearAxisZ.commandConfiguration.phasing.direction := 3;
   cmMendrelCathodeRearAxisZ.commandConfiguration.phasing.phaseAbsolute := TRUE;
   cmMendrelCathodeRearAxisZ.commandConfiguration.phasing.phaseShiftChangeOnTheFly := FALSE;
   cmMendrelCathodeRearAxisZ.commandConfiguration.offset.offset := 0.0;
   cmMendrelCathodeRearAxisZ.commandConfiguration.offset.profileReference := 1;
   cmMendrelCathodeRearAxisZ.commandConfiguration.offset.offsetDistance := 0.0;
   cmMendrelCathodeRearAxisZ.commandConfiguration.offset.startPosition := 0.0;
   cmMendrelCathodeRearAxisZ.commandConfiguration.offset.direction := 3;
   cmMendrelCathodeRearAxisZ.commandConfiguration.offset.offsetAbsolute := TRUE;
   cmMendrelCathodeRearAxisZ.commandConfiguration.offset.offsetChangeOnTheFly := FALSE;
   cmMendrelCathodeRearAxisZ.commands.enableMasterControl := TRUE;
   cmMendrelCathodeRearAxisZ.commands.enableAxis := FALSE;
   cmMendrelCathodeRearAxisZ.commands.resetAxis := FALSE;
   cmMendrelCathodeRearAxisZ.commands.openBrake := FALSE;
   cmMendrelCathodeRearAxisZ.commands.jogForward := FALSE;
   cmMendrelCathodeRearAxisZ.commands.jogBackward := FALSE;
   cmMendrelCathodeRearAxisZ.commands.moveVelocity := FALSE;
   cmMendrelCathodeRearAxisZ.commands.stop := FALSE;
   cmMendrelCathodeRearAxisZ.commands.fastStop := FALSE;
   cmMendrelCathodeRearAxisZ.commands.torqueLimiting := FALSE;
   cmMendrelCathodeRearAxisZ.commands.homing := FALSE;
   cmMendrelCathodeRearAxisZ.commands.posRelative := FALSE;
   cmMendrelCathodeRearAxisZ.commands.posAbsolute := FALSE;
   cmMendrelCathodeRearAxisZ.commands.posSuperimposed := FALSE;
   cmMendrelCathodeRearAxisZ.commands.haltSuperimposed := FALSE;
   cmMendrelCathodeRearAxisZ.commands.selectSetPosition := 1;
   cmMendrelCathodeRearAxisZ.commands.uploadParameters := FALSE;
   cmMendrelCathodeRearAxisZ.commands.refreshConfiguration := FALSE;
   cmMendrelCathodeRearAxisZ.commands.editConfiguration := FALSE;
   cmMendrelCathodeRearAxisZ.commands.saveConfiguration := FALSE;
   cmMendrelCathodeRearAxisZ.commands.uploadCurrentTorque := FALSE;
   cmMendrelCathodeRearAxisZ.commands.reset := FALSE;
   cmMendrelCathodeRearAxisZ.monitoring.enable := TRUE;
   cmMendrelCathodeRearAxisZ.monitoring.referenceDesignator := WSTRING#'MendrelCathodeRearAxisZ';
   cmMendrelCathodeRearAxisZ.monitoring.enabled := TRUE;
   cmMendrelCathodeRearAxisZ.monitoring.enableManualCmds := FALSE;
   cmMendrelCathodeRearAxisZ.monitoring.reset := FALSE;
   cmMendrelCathodeRearAxisZ.monitoring.resetAxis := FALSE;
   cmMendrelCathodeRearAxisZ.monitoring.enableAxis := TRUE;
   cmMendrelCathodeRearAxisZ.monitoring.openBrake := FALSE;
   cmMendrelCathodeRearAxisZ.monitoring.jogBackward := FALSE;
   cmMendrelCathodeRearAxisZ.monitoring.jogForward := FALSE;
   cmMendrelCathodeRearAxisZ.monitoring.moveVelocity := FALSE;
   cmMendrelCathodeRearAxisZ.monitoring.stop := FALSE;
   cmMendrelCathodeRearAxisZ.monitoring.fastStop := FALSE;
   cmMendrelCathodeRearAxisZ.monitoring.torqueLimiting := FALSE;
   cmMendrelCathodeRearAxisZ.monitoring.homing := FALSE;
   cmMendrelCathodeRearAxisZ.monitoring.posRelative := FALSE;
   cmMendrelCathodeRearAxisZ.monitoring.posAbsolute := FALSE;
   cmMendrelCathodeRearAxisZ.monitoring.posSuperimposed := FALSE;
   cmMendrelCathodeRearAxisZ.monitoring.haltSuperimposed := FALSE;
   cmMendrelCathodeRearAxisZ.monitoring.brakeOpened := FALSE;
   cmMendrelCathodeRearAxisZ.monitoring.axisEnabled := TRUE;
   cmMendrelCathodeRearAxisZ.monitoring.resetActive := FALSE;
   cmMendrelCathodeRearAxisZ.monitoring.inVelocity := FALSE;
   cmMendrelCathodeRearAxisZ.monitoring.inLimitation := FALSE;
   cmMendrelCathodeRearAxisZ.monitoring.inClamping := FALSE;
   cmMendrelCathodeRearAxisZ.monitoring.startSync := FALSE;
   cmMendrelCathodeRearAxisZ.monitoring.inSync := FALSE;
   cmMendrelCathodeRearAxisZ.monitoring.inSimulation := FALSE;
   cmMendrelCathodeRearAxisZ.monitoring.jogSelected := FALSE;
   cmMendrelCathodeRearAxisZ.monitoring.moveVelocitySelected := FALSE;
   cmMendrelCathodeRearAxisZ.monitoring.stopSelected := FALSE;
   cmMendrelCathodeRearAxisZ.monitoring.fastStopSelected := FALSE;
   cmMendrelCathodeRearAxisZ.monitoring.torqueLimitingSelected := FALSE;
   cmMendrelCathodeRearAxisZ.monitoring.homingSelected := FALSE;
   cmMendrelCathodeRearAxisZ.monitoring.posRelativeSelected := FALSE;
   cmMendrelCathodeRearAxisZ.monitoring.posAbsoluteSelected := FALSE;
   cmMendrelCathodeRearAxisZ.monitoring.posSuperimposedSelected := FALSE;
   cmMendrelCathodeRearAxisZ.monitoring.haltSuperimposedSelected := FALSE;
   cmMendrelCathodeRearAxisZ.monitoring.commandBusy := FALSE;
   cmMendrelCathodeRearAxisZ.monitoring.commandDone := FALSE;
   cmMendrelCathodeRearAxisZ.monitoring.commandAborted := FALSE;
   cmMendrelCathodeRearAxisZ.monitoring.homingCommandBusy := FALSE;
   cmMendrelCathodeRearAxisZ.monitoring.homingCommandDone := FALSE;
   cmMendrelCathodeRearAxisZ.monitoring.homingCommandAborted := FALSE;
   cmMendrelCathodeRearAxisZ.monitoring.superimposedBusy := FALSE;
   cmMendrelCathodeRearAxisZ.monitoring.superimposedDone := FALSE;
   cmMendrelCathodeRearAxisZ.monitoring.superimposedAborted := FALSE;
   cmMendrelCathodeRearAxisZ.monitoring.selectSetPosition := 1;
   cmMendrelCathodeRearAxisZ.monitoring.selectionController := FALSE;
   cmMendrelCathodeRearAxisZ.monitoring.interlockGeneral := TRUE;
   cmMendrelCathodeRearAxisZ.monitoring.interlockJogForward := TRUE;
   cmMendrelCathodeRearAxisZ.monitoring.interlockJogBackward := TRUE;
   cmMendrelCathodeRearAxisZ.monitoring.interlockWarningGeneral := FALSE;
   cmMendrelCathodeRearAxisZ.monitoring.interlockWarningJogForward := FALSE;
   cmMendrelCathodeRearAxisZ.monitoring.interlockWarningJogBackward := FALSE;
   cmMendrelCathodeRearAxisZ.monitoring.valid := TRUE;
   cmMendrelCathodeRearAxisZ.monitoring.busy := TRUE;
   cmMendrelCathodeRearAxisZ.monitoring.error := FALSE;
   cmMendrelCathodeRearAxisZ.monitoring.status := 16#7002;
   cmMendrelCathodeRearAxisZ.monitoring.subfunctionStatus := 16#0000;
   cmMendrelCathodeRearAxisZ.monitoring.actualPosition := 0.0;
   cmMendrelCathodeRearAxisZ.monitoring.actualSpeed := 0.0;
   cmMendrelCathodeRearAxisZ.monitoring.speedUnit := 1062;
   cmMendrelCathodeRearAxisZ.monitoring.positionUnit := 1013;
   cmMendrelCathodeRearAxisZ.monitoring.axisStatus1 := 16#0240_10A1;
   cmMendrelCathodeRearAxisZ.monitoring.axisStatus2 := 16#0000_0000;
   cmMendrelCathodeRearAxisZ.monitoring.axisType := 1;
   cmMendrelCathodeRearAxisZ.monitoring.maxVelocity := 2500.0;
   cmMendrelCathodeRearAxisZ.monitoring.actualCurrent := 0.0;
   cmMendrelCathodeRearAxisZ.monitoring.actualTorque := 0.0;
   cmMendrelCathodeRearAxisZ.monitoring.velocityOverrideEnabled := FALSE;
   cmMendrelCathodeRearAxisZ.monitoring.sinaParaError := FALSE;
   cmMendrelCathodeRearAxisZ.monitoring.sinaParaStatus := 16#0000_0000;
   cmMendrelCathodeRearAxisZ.configuration.referenceDesignator := WSTRING#'MendrelCathodeRearAxisZ';
   cmMendrelCathodeRearAxisZ.configuration.disableAlarms := FALSE;
   cmMendrelCathodeRearAxisZ.configuration.masterControlPopUp := TRUE;
   cmMendrelCathodeRearAxisZ.configuration.setPositions[0].position := 0.0;
   cmMendrelCathodeRearAxisZ.configuration.setPositions[1].position := 50.0;
   cmMendrelCathodeRearAxisZ.configuration.setPositions[2..15].position := 0.0;
   cmMendrelCathodeRearAxisZ.configuration.setPositions[0..1].velocity := 50.0;
   cmMendrelCathodeRearAxisZ.configuration.setPositions[2..15].velocity := -1.0;
   cmMendrelCathodeRearAxisZ.configuration.setPositions[0..1].acceleration := 500.0;
   cmMendrelCathodeRearAxisZ.configuration.setPositions[2..15].acceleration := -1.0;
   cmMendrelCathodeRearAxisZ.configuration.setPositions[0..1].deceleration := 500.0;
   cmMendrelCathodeRearAxisZ.configuration.setPositions[2..15].deceleration := -1.0;
   cmMendrelCathodeRearAxisZ.configuration.setPositions[0..15]."name" := '';
   cmStackTableAxisZ.commandConfiguration.generalSettings.stopOnError := TRUE;
   cmStackTableAxisZ.commandConfiguration.generalSettings.resetWithRestart := FALSE;
   cmStackTableAxisZ.commandConfiguration.generalSettings.abortWaitingSyncCmd := TRUE;
   cmStackTableAxisZ.commandConfiguration.power.startMode := 1;
   cmStackTableAxisZ.commandConfiguration.power.stopMode := 0;
   cmStackTableAxisZ.commandConfiguration.power.syncMotionSimulation := FALSE;
   cmStackTableAxisZ.commandConfiguration.power.syncMotionSimulationExtendedMode := -1;
   cmStackTableAxisZ.commandConfiguration.jog.velocity := 0.0;
   cmStackTableAxisZ.commandConfiguration.jog.acceleration := -1.0;
   cmStackTableAxisZ.commandConfiguration.jog.deceleration := -1.0;
   cmStackTableAxisZ.commandConfiguration.jog.jerk := -1.0;
   cmStackTableAxisZ.commandConfiguration.jog.positionControlled := TRUE;
   cmStackTableAxisZ.commandConfiguration.jog.increment := 0.0;
   cmStackTableAxisZ.commandConfiguration.jog.mode := 0;
   cmStackTableAxisZ.commandConfiguration.moveVelocity.velocity := 0.0;
   cmStackTableAxisZ.commandConfiguration.moveVelocity.acceleration := -1.0;
   cmStackTableAxisZ.commandConfiguration.moveVelocity.deceleration := -1.0;
   cmStackTableAxisZ.commandConfiguration.moveVelocity.jerk := -1.0;
   cmStackTableAxisZ.commandConfiguration.moveVelocity.direction := 0;
   cmStackTableAxisZ.commandConfiguration.moveVelocity.positionControlled := TRUE;
   cmStackTableAxisZ.commandConfiguration.moveVelocity.velocityChangeOnTheFly := FALSE;
   cmStackTableAxisZ.commandConfiguration.stop.deceleration := -1.0;
   cmStackTableAxisZ.commandConfiguration.stop.jerk := -1.0;
   cmStackTableAxisZ.commandConfiguration.stop.abortAcceleration := FALSE;
   cmStackTableAxisZ.commandConfiguration.fastStop.deceleration := -1.0;
   cmStackTableAxisZ.commandConfiguration.fastStop.jerk := -1.0;
   cmStackTableAxisZ.commandConfiguration.fastStop.abortAcceleration := FALSE;
   cmStackTableAxisZ.commandConfiguration.fastStop.replaceStopPossible := FALSE;
   cmStackTableAxisZ.commandConfiguration.torqueLimiting.limit := -1.0;
   cmStackTableAxisZ.commandConfiguration.torqueLimiting.mode := 0;
   cmStackTableAxisZ.commandConfiguration.homing.position := 0.0;
   cmStackTableAxisZ.commandConfiguration.homing.mode := 0;
   cmStackTableAxisZ.commandConfiguration.homing.sensor := 0;
   cmStackTableAxisZ.commandConfiguration.homing.extendedMode := -1;
   cmStackTableAxisZ.commandConfiguration.homing.extendedModeTorqueLimit := 0.0;
   cmStackTableAxisZ.commandConfiguration.homing.extendedModeTargetPosition := 0.0;
   cmStackTableAxisZ.commandConfiguration.posRelative.distance := 0.0;
   cmStackTableAxisZ.commandConfiguration.posRelative.velocity := -1.0;
   cmStackTableAxisZ.commandConfiguration.posRelative.acceleration := -1.0;
   cmStackTableAxisZ.commandConfiguration.posRelative.deceleration := -1.0;
   cmStackTableAxisZ.commandConfiguration.posRelative.jerk := -1.0;
   cmStackTableAxisZ.commandConfiguration.posRelative.direction := 0;
   cmStackTableAxisZ.commandConfiguration.posAbsolute.position := 0.0;
   cmStackTableAxisZ.commandConfiguration.posAbsolute.velocity := -1.0;
   cmStackTableAxisZ.commandConfiguration.posAbsolute.acceleration := -1.0;
   cmStackTableAxisZ.commandConfiguration.posAbsolute.deceleration := -1.0;
   cmStackTableAxisZ.commandConfiguration.posAbsolute.jerk := -1.0;
   cmStackTableAxisZ.commandConfiguration.posAbsolute.direction := 1;
   cmStackTableAxisZ.commandConfiguration.posAbsolute.positionChangeOnTheFly := FALSE;
   cmStackTableAxisZ.commandConfiguration.posAbsolute.velocityChangeOnTheFly := FALSE;
   cmStackTableAxisZ.commandConfiguration.posSuperimposed.distance := 0.0;
   cmStackTableAxisZ.commandConfiguration.posSuperimposed.velocityDiff := -1.0;
   cmStackTableAxisZ.commandConfiguration.posSuperimposed.acceleration := -1.0;
   cmStackTableAxisZ.commandConfiguration.posSuperimposed.deceleration := -1.0;
   cmStackTableAxisZ.commandConfiguration.posSuperimposed.jerk := -1.0;
   cmStackTableAxisZ.commandConfiguration.posSuperimposed.direction := 0;
   cmStackTableAxisZ.commandConfiguration.haltSuperimposed.deceleration := -1.0;
   cmStackTableAxisZ.commandConfiguration.haltSuperimposed.jerk := -1.0;
   cmStackTableAxisZ.commandConfiguration.haltSuperimposed.abortAcceleration := FALSE;
   cmStackTableAxisZ.commandConfiguration.gearInRelative.ratioNumerator := 1;
   cmStackTableAxisZ.commandConfiguration.gearInRelative.ratioDenominator := 1;
   cmStackTableAxisZ.commandConfiguration.gearInRelative.acceleration := -1.0;
   cmStackTableAxisZ.commandConfiguration.gearInRelative.deceleration := -1.0;
   cmStackTableAxisZ.commandConfiguration.gearInRelative.jerk := -1.0;
   cmStackTableAxisZ.commandConfiguration.gearInRelative.ratioChangeOnTheFly := FALSE;
   cmStackTableAxisZ.commandConfiguration.gearInAbsolute.ratioNumerator := 1;
   cmStackTableAxisZ.commandConfiguration.gearInAbsolute.ratioDenominator := 1;
   cmStackTableAxisZ.commandConfiguration.gearInAbsolute.masterSyncPosition := 0.0;
   cmStackTableAxisZ.commandConfiguration.gearInAbsolute.slaveSyncPosition := 0.0;
   cmStackTableAxisZ.commandConfiguration.gearInAbsolute.syncProfileReference := 1;
   cmStackTableAxisZ.commandConfiguration.gearInAbsolute.masterStartDistance := 0.0;
   cmStackTableAxisZ.commandConfiguration.gearInAbsolute.velocity := -1.0;
   cmStackTableAxisZ.commandConfiguration.gearInAbsolute.acceleration := -1.0;
   cmStackTableAxisZ.commandConfiguration.gearInAbsolute.deceleration := -1.0;
   cmStackTableAxisZ.commandConfiguration.gearInAbsolute.jerk := -1.0;
   cmStackTableAxisZ.commandConfiguration.gearInAbsolute.syncDirection := 1;
   cmStackTableAxisZ.commandConfiguration.gearInAbsolute.ratioChangeOnTheFly := FALSE;
   cmStackTableAxisZ.commandConfiguration.gearInVelocity.continuousUpdate := FALSE;
   cmStackTableAxisZ.commandConfiguration.gearInVelocity.ratioNumerator := 1;
   cmStackTableAxisZ.commandConfiguration.gearInVelocity.ratioDenominator := 1;
   cmStackTableAxisZ.commandConfiguration.gearInVelocity.acceleration := -1.0;
   cmStackTableAxisZ.commandConfiguration.gearInVelocity.deceleration := -1.0;
   cmStackTableAxisZ.commandConfiguration.gearInVelocity.jerk := -1.0;
   cmStackTableAxisZ.commandConfiguration.gearInVelocity.positionControlled := FALSE;
   cmStackTableAxisZ.commandConfiguration.camIn.masterOffset := 0.0;
   cmStackTableAxisZ.commandConfiguration.camIn.slaveOffset := 0.0;
   cmStackTableAxisZ.commandConfiguration.camIn.masterScaling := 1.0;
   cmStackTableAxisZ.commandConfiguration.camIn.slaveScaling := 1.0;
   cmStackTableAxisZ.commandConfiguration.camIn.masterSyncPosition := 0.0;
   cmStackTableAxisZ.commandConfiguration.camIn.syncProfileReference := 1;
   cmStackTableAxisZ.commandConfiguration.camIn.masterStartDistance := 0.0;
   cmStackTableAxisZ.commandConfiguration.camIn.velocity := -1.0;
   cmStackTableAxisZ.commandConfiguration.camIn.acceleration := -1.0;
   cmStackTableAxisZ.commandConfiguration.camIn.deceleration := -1.0;
   cmStackTableAxisZ.commandConfiguration.camIn.jerk := -1.0;
   cmStackTableAxisZ.commandConfiguration.camIn.applicationMode := 0;
   cmStackTableAxisZ.commandConfiguration.camIn.syncDirection := 1;
   cmStackTableAxisZ.commandConfiguration.gearOutCamOut.slavePosition := 0.0;
   cmStackTableAxisZ.commandConfiguration.gearOutCamOut.syncProfileReference := 1;
   cmStackTableAxisZ.commandConfiguration.gearOutCamOut.masterStopDistance := 0.0;
   cmStackTableAxisZ.commandConfiguration.gearOutCamOut.deceleration := -1.0;
   cmStackTableAxisZ.commandConfiguration.gearOutCamOut.jerk := -1.0;
   cmStackTableAxisZ.commandConfiguration.gearOutCamOut.syncOutDirection := 3;
   cmStackTableAxisZ.commandConfiguration.gearOutCamOut.gearOutCamOutMode := -1;
   cmStackTableAxisZ.commandConfiguration.phasing.phaseShift := 0.0;
   cmStackTableAxisZ.commandConfiguration.phasing.velocity := -1.0;
   cmStackTableAxisZ.commandConfiguration.phasing.acceleration := -1.0;
   cmStackTableAxisZ.commandConfiguration.phasing.deceleration := -1.0;
   cmStackTableAxisZ.commandConfiguration.phasing.jerk := -1.0;
   cmStackTableAxisZ.commandConfiguration.phasing.profileReference := 0;
   cmStackTableAxisZ.commandConfiguration.phasing.phasingDistance := 0.0;
   cmStackTableAxisZ.commandConfiguration.phasing.startPosition := 0.0;
   cmStackTableAxisZ.commandConfiguration.phasing.direction := 3;
   cmStackTableAxisZ.commandConfiguration.phasing.phaseAbsolute := TRUE;
   cmStackTableAxisZ.commandConfiguration.phasing.phaseShiftChangeOnTheFly := FALSE;
   cmStackTableAxisZ.commandConfiguration.offset.offset := 0.0;
   cmStackTableAxisZ.commandConfiguration.offset.profileReference := 1;
   cmStackTableAxisZ.commandConfiguration.offset.offsetDistance := 0.0;
   cmStackTableAxisZ.commandConfiguration.offset.startPosition := 0.0;
   cmStackTableAxisZ.commandConfiguration.offset.direction := 3;
   cmStackTableAxisZ.commandConfiguration.offset.offsetAbsolute := TRUE;
   cmStackTableAxisZ.commandConfiguration.offset.offsetChangeOnTheFly := FALSE;
   cmStackTableAxisZ.commands.enableMasterControl := TRUE;
   cmStackTableAxisZ.commands.enableAxis := FALSE;
   cmStackTableAxisZ.commands.resetAxis := FALSE;
   cmStackTableAxisZ.commands.openBrake := FALSE;
   cmStackTableAxisZ.commands.jogForward := FALSE;
   cmStackTableAxisZ.commands.jogBackward := FALSE;
   cmStackTableAxisZ.commands.moveVelocity := FALSE;
   cmStackTableAxisZ.commands.stop := FALSE;
   cmStackTableAxisZ.commands.fastStop := FALSE;
   cmStackTableAxisZ.commands.torqueLimiting := FALSE;
   cmStackTableAxisZ.commands.homing := FALSE;
   cmStackTableAxisZ.commands.posRelative := FALSE;
   cmStackTableAxisZ.commands.posAbsolute := FALSE;
   cmStackTableAxisZ.commands.posSuperimposed := FALSE;
   cmStackTableAxisZ.commands.haltSuperimposed := FALSE;
   cmStackTableAxisZ.commands.selectSetPosition := -1;
   cmStackTableAxisZ.commands.uploadParameters := FALSE;
   cmStackTableAxisZ.commands.refreshConfiguration := FALSE;
   cmStackTableAxisZ.commands.editConfiguration := FALSE;
   cmStackTableAxisZ.commands.saveConfiguration := FALSE;
   cmStackTableAxisZ.commands.uploadCurrentTorque := FALSE;
   cmStackTableAxisZ.commands.reset := FALSE;
   cmStackTableAxisZ.monitoring.enable := TRUE;
   cmStackTableAxisZ.monitoring.referenceDesignator := WSTRING#'StackTableAxisZ';
   cmStackTableAxisZ.monitoring.enabled := TRUE;
   cmStackTableAxisZ.monitoring.enableManualCmds := FALSE;
   cmStackTableAxisZ.monitoring.reset := FALSE;
   cmStackTableAxisZ.monitoring.resetAxis := FALSE;
   cmStackTableAxisZ.monitoring.enableAxis := TRUE;
   cmStackTableAxisZ.monitoring.openBrake := FALSE;
   cmStackTableAxisZ.monitoring.jogBackward := FALSE;
   cmStackTableAxisZ.monitoring.jogForward := FALSE;
   cmStackTableAxisZ.monitoring.moveVelocity := FALSE;
   cmStackTableAxisZ.monitoring.stop := FALSE;
   cmStackTableAxisZ.monitoring.fastStop := FALSE;
   cmStackTableAxisZ.monitoring.torqueLimiting := FALSE;
   cmStackTableAxisZ.monitoring.homing := FALSE;
   cmStackTableAxisZ.monitoring.posRelative := FALSE;
   cmStackTableAxisZ.monitoring.posAbsolute := FALSE;
   cmStackTableAxisZ.monitoring.posSuperimposed := FALSE;
   cmStackTableAxisZ.monitoring.haltSuperimposed := FALSE;
   cmStackTableAxisZ.monitoring.brakeOpened := FALSE;
   cmStackTableAxisZ.monitoring.axisEnabled := TRUE;
   cmStackTableAxisZ.monitoring.resetActive := FALSE;
   cmStackTableAxisZ.monitoring.inVelocity := FALSE;
   cmStackTableAxisZ.monitoring.inLimitation := FALSE;
   cmStackTableAxisZ.monitoring.inClamping := FALSE;
   cmStackTableAxisZ.monitoring.startSync := FALSE;
   cmStackTableAxisZ.monitoring.inSync := FALSE;
   cmStackTableAxisZ.monitoring.inSimulation := FALSE;
   cmStackTableAxisZ.monitoring.jogSelected := FALSE;
   cmStackTableAxisZ.monitoring.moveVelocitySelected := FALSE;
   cmStackTableAxisZ.monitoring.stopSelected := FALSE;
   cmStackTableAxisZ.monitoring.fastStopSelected := FALSE;
   cmStackTableAxisZ.monitoring.torqueLimitingSelected := FALSE;
   cmStackTableAxisZ.monitoring.homingSelected := FALSE;
   cmStackTableAxisZ.monitoring.posRelativeSelected := FALSE;
   cmStackTableAxisZ.monitoring.posAbsoluteSelected := FALSE;
   cmStackTableAxisZ.monitoring.posSuperimposedSelected := FALSE;
   cmStackTableAxisZ.monitoring.haltSuperimposedSelected := FALSE;
   cmStackTableAxisZ.monitoring.commandBusy := FALSE;
   cmStackTableAxisZ.monitoring.commandDone := FALSE;
   cmStackTableAxisZ.monitoring.commandAborted := FALSE;
   cmStackTableAxisZ.monitoring.homingCommandBusy := FALSE;
   cmStackTableAxisZ.monitoring.homingCommandDone := FALSE;
   cmStackTableAxisZ.monitoring.homingCommandAborted := FALSE;
   cmStackTableAxisZ.monitoring.superimposedBusy := FALSE;
   cmStackTableAxisZ.monitoring.superimposedDone := FALSE;
   cmStackTableAxisZ.monitoring.superimposedAborted := FALSE;
   cmStackTableAxisZ.monitoring.selectSetPosition := -1;
   cmStackTableAxisZ.monitoring.selectionController := FALSE;
   cmStackTableAxisZ.monitoring.interlockGeneral := TRUE;
   cmStackTableAxisZ.monitoring.interlockJogForward := TRUE;
   cmStackTableAxisZ.monitoring.interlockJogBackward := TRUE;
   cmStackTableAxisZ.monitoring.interlockWarningGeneral := FALSE;
   cmStackTableAxisZ.monitoring.interlockWarningJogForward := FALSE;
   cmStackTableAxisZ.monitoring.interlockWarningJogBackward := FALSE;
   cmStackTableAxisZ.monitoring.valid := TRUE;
   cmStackTableAxisZ.monitoring.busy := TRUE;
   cmStackTableAxisZ.monitoring.error := FALSE;
   cmStackTableAxisZ.monitoring.status := 16#7002;
   cmStackTableAxisZ.monitoring.subfunctionStatus := 16#0000;
   cmStackTableAxisZ.monitoring.actualPosition := 0.0;
   cmStackTableAxisZ.monitoring.actualSpeed := 0.0;
   cmStackTableAxisZ.monitoring.speedUnit := 1062;
   cmStackTableAxisZ.monitoring.positionUnit := 1013;
   cmStackTableAxisZ.monitoring.axisStatus1 := 16#0200_10E1;
   cmStackTableAxisZ.monitoring.axisStatus2 := 16#0000_0000;
   cmStackTableAxisZ.monitoring.axisType := 1;
   cmStackTableAxisZ.monitoring.maxVelocity := 2500.0;
   cmStackTableAxisZ.monitoring.actualCurrent := 0.0;
   cmStackTableAxisZ.monitoring.actualTorque := 0.0;
   cmStackTableAxisZ.monitoring.velocityOverrideEnabled := FALSE;
   cmStackTableAxisZ.monitoring.sinaParaError := FALSE;
   cmStackTableAxisZ.monitoring.sinaParaStatus := 16#0000_0000;
   cmStackTableAxisZ.configuration.referenceDesignator := WSTRING#'StackTableAxisZ';
   cmStackTableAxisZ.configuration.disableAlarms := FALSE;
   cmStackTableAxisZ.configuration.masterControlPopUp := TRUE;
   cmStackTableAxisZ.configuration.setPositions[0].position := 50.0;
   cmStackTableAxisZ.configuration.setPositions[1..15].position := 0.0;
   cmStackTableAxisZ.configuration.setPositions[0..1].velocity := 50.0;
   cmStackTableAxisZ.configuration.setPositions[2..15].velocity := -1.0;
   cmStackTableAxisZ.configuration.setPositions[0..1].acceleration := 500.0;
   cmStackTableAxisZ.configuration.setPositions[2..15].acceleration := -1.0;
   cmStackTableAxisZ.configuration.setPositions[0..1].deceleration := 500.0;
   cmStackTableAxisZ.configuration.setPositions[2..15].deceleration := -1.0;
   cmStackTableAxisZ.configuration.setPositions[0..15]."name" := '';
   cmStackTableOutFrontAxisZ.commandConfiguration.generalSettings.stopOnError := TRUE;
   cmStackTableOutFrontAxisZ.commandConfiguration.generalSettings.resetWithRestart := FALSE;
   cmStackTableOutFrontAxisZ.commandConfiguration.generalSettings.abortWaitingSyncCmd := TRUE;
   cmStackTableOutFrontAxisZ.commandConfiguration.power.startMode := 1;
   cmStackTableOutFrontAxisZ.commandConfiguration.power.stopMode := 0;
   cmStackTableOutFrontAxisZ.commandConfiguration.power.syncMotionSimulation := FALSE;
   cmStackTableOutFrontAxisZ.commandConfiguration.power.syncMotionSimulationExtendedMode := -1;
   cmStackTableOutFrontAxisZ.commandConfiguration.jog.velocity := 0.0;
   cmStackTableOutFrontAxisZ.commandConfiguration.jog.acceleration := -1.0;
   cmStackTableOutFrontAxisZ.commandConfiguration.jog.deceleration := -1.0;
   cmStackTableOutFrontAxisZ.commandConfiguration.jog.jerk := -1.0;
   cmStackTableOutFrontAxisZ.commandConfiguration.jog.positionControlled := TRUE;
   cmStackTableOutFrontAxisZ.commandConfiguration.jog.increment := 0.0;
   cmStackTableOutFrontAxisZ.commandConfiguration.jog.mode := 0;
   cmStackTableOutFrontAxisZ.commandConfiguration.moveVelocity.velocity := 0.0;
   cmStackTableOutFrontAxisZ.commandConfiguration.moveVelocity.acceleration := -1.0;
   cmStackTableOutFrontAxisZ.commandConfiguration.moveVelocity.deceleration := -1.0;
   cmStackTableOutFrontAxisZ.commandConfiguration.moveVelocity.jerk := -1.0;
   cmStackTableOutFrontAxisZ.commandConfiguration.moveVelocity.direction := 0;
   cmStackTableOutFrontAxisZ.commandConfiguration.moveVelocity.positionControlled := TRUE;
   cmStackTableOutFrontAxisZ.commandConfiguration.moveVelocity.velocityChangeOnTheFly := FALSE;
   cmStackTableOutFrontAxisZ.commandConfiguration.stop.deceleration := -1.0;
   cmStackTableOutFrontAxisZ.commandConfiguration.stop.jerk := -1.0;
   cmStackTableOutFrontAxisZ.commandConfiguration.stop.abortAcceleration := FALSE;
   cmStackTableOutFrontAxisZ.commandConfiguration.fastStop.deceleration := -1.0;
   cmStackTableOutFrontAxisZ.commandConfiguration.fastStop.jerk := -1.0;
   cmStackTableOutFrontAxisZ.commandConfiguration.fastStop.abortAcceleration := FALSE;
   cmStackTableOutFrontAxisZ.commandConfiguration.fastStop.replaceStopPossible := FALSE;
   cmStackTableOutFrontAxisZ.commandConfiguration.torqueLimiting.limit := -1.0;
   cmStackTableOutFrontAxisZ.commandConfiguration.torqueLimiting.mode := 0;
   cmStackTableOutFrontAxisZ.commandConfiguration.homing.position := 0.0;
   cmStackTableOutFrontAxisZ.commandConfiguration.homing.mode := 0;
   cmStackTableOutFrontAxisZ.commandConfiguration.homing.sensor := 0;
   cmStackTableOutFrontAxisZ.commandConfiguration.homing.extendedMode := -1;
   cmStackTableOutFrontAxisZ.commandConfiguration.homing.extendedModeTorqueLimit := 0.0;
   cmStackTableOutFrontAxisZ.commandConfiguration.homing.extendedModeTargetPosition := 0.0;
   cmStackTableOutFrontAxisZ.commandConfiguration.posRelative.distance := 0.0;
   cmStackTableOutFrontAxisZ.commandConfiguration.posRelative.velocity := -1.0;
   cmStackTableOutFrontAxisZ.commandConfiguration.posRelative.acceleration := -1.0;
   cmStackTableOutFrontAxisZ.commandConfiguration.posRelative.deceleration := -1.0;
   cmStackTableOutFrontAxisZ.commandConfiguration.posRelative.jerk := -1.0;
   cmStackTableOutFrontAxisZ.commandConfiguration.posRelative.direction := 0;
   cmStackTableOutFrontAxisZ.commandConfiguration.posAbsolute.position := 0.0;
   cmStackTableOutFrontAxisZ.commandConfiguration.posAbsolute.velocity := -1.0;
   cmStackTableOutFrontAxisZ.commandConfiguration.posAbsolute.acceleration := -1.0;
   cmStackTableOutFrontAxisZ.commandConfiguration.posAbsolute.deceleration := -1.0;
   cmStackTableOutFrontAxisZ.commandConfiguration.posAbsolute.jerk := -1.0;
   cmStackTableOutFrontAxisZ.commandConfiguration.posAbsolute.direction := 1;
   cmStackTableOutFrontAxisZ.commandConfiguration.posAbsolute.positionChangeOnTheFly := FALSE;
   cmStackTableOutFrontAxisZ.commandConfiguration.posAbsolute.velocityChangeOnTheFly := FALSE;
   cmStackTableOutFrontAxisZ.commandConfiguration.posSuperimposed.distance := 0.0;
   cmStackTableOutFrontAxisZ.commandConfiguration.posSuperimposed.velocityDiff := -1.0;
   cmStackTableOutFrontAxisZ.commandConfiguration.posSuperimposed.acceleration := -1.0;
   cmStackTableOutFrontAxisZ.commandConfiguration.posSuperimposed.deceleration := -1.0;
   cmStackTableOutFrontAxisZ.commandConfiguration.posSuperimposed.jerk := -1.0;
   cmStackTableOutFrontAxisZ.commandConfiguration.posSuperimposed.direction := 0;
   cmStackTableOutFrontAxisZ.commandConfiguration.haltSuperimposed.deceleration := -1.0;
   cmStackTableOutFrontAxisZ.commandConfiguration.haltSuperimposed.jerk := -1.0;
   cmStackTableOutFrontAxisZ.commandConfiguration.haltSuperimposed.abortAcceleration := FALSE;
   cmStackTableOutFrontAxisZ.commandConfiguration.gearInRelative.ratioNumerator := 1;
   cmStackTableOutFrontAxisZ.commandConfiguration.gearInRelative.ratioDenominator := 1;
   cmStackTableOutFrontAxisZ.commandConfiguration.gearInRelative.acceleration := -1.0;
   cmStackTableOutFrontAxisZ.commandConfiguration.gearInRelative.deceleration := -1.0;
   cmStackTableOutFrontAxisZ.commandConfiguration.gearInRelative.jerk := -1.0;
   cmStackTableOutFrontAxisZ.commandConfiguration.gearInRelative.ratioChangeOnTheFly := FALSE;
   cmStackTableOutFrontAxisZ.commandConfiguration.gearInAbsolute.ratioNumerator := 1;
   cmStackTableOutFrontAxisZ.commandConfiguration.gearInAbsolute.ratioDenominator := 1;
   cmStackTableOutFrontAxisZ.commandConfiguration.gearInAbsolute.masterSyncPosition := 0.0;
   cmStackTableOutFrontAxisZ.commandConfiguration.gearInAbsolute.slaveSyncPosition := 0.0;
   cmStackTableOutFrontAxisZ.commandConfiguration.gearInAbsolute.syncProfileReference := 1;
   cmStackTableOutFrontAxisZ.commandConfiguration.gearInAbsolute.masterStartDistance := 0.0;
   cmStackTableOutFrontAxisZ.commandConfiguration.gearInAbsolute.velocity := -1.0;
   cmStackTableOutFrontAxisZ.commandConfiguration.gearInAbsolute.acceleration := -1.0;
   cmStackTableOutFrontAxisZ.commandConfiguration.gearInAbsolute.deceleration := -1.0;
   cmStackTableOutFrontAxisZ.commandConfiguration.gearInAbsolute.jerk := -1.0;
   cmStackTableOutFrontAxisZ.commandConfiguration.gearInAbsolute.syncDirection := 1;
   cmStackTableOutFrontAxisZ.commandConfiguration.gearInAbsolute.ratioChangeOnTheFly := FALSE;
   cmStackTableOutFrontAxisZ.commandConfiguration.gearInVelocity.continuousUpdate := FALSE;
   cmStackTableOutFrontAxisZ.commandConfiguration.gearInVelocity.ratioNumerator := 1;
   cmStackTableOutFrontAxisZ.commandConfiguration.gearInVelocity.ratioDenominator := 1;
   cmStackTableOutFrontAxisZ.commandConfiguration.gearInVelocity.acceleration := -1.0;
   cmStackTableOutFrontAxisZ.commandConfiguration.gearInVelocity.deceleration := -1.0;
   cmStackTableOutFrontAxisZ.commandConfiguration.gearInVelocity.jerk := -1.0;
   cmStackTableOutFrontAxisZ.commandConfiguration.gearInVelocity.positionControlled := FALSE;
   cmStackTableOutFrontAxisZ.commandConfiguration.camIn.masterOffset := 0.0;
   cmStackTableOutFrontAxisZ.commandConfiguration.camIn.slaveOffset := 0.0;
   cmStackTableOutFrontAxisZ.commandConfiguration.camIn.masterScaling := 1.0;
   cmStackTableOutFrontAxisZ.commandConfiguration.camIn.slaveScaling := 1.0;
   cmStackTableOutFrontAxisZ.commandConfiguration.camIn.masterSyncPosition := 0.0;
   cmStackTableOutFrontAxisZ.commandConfiguration.camIn.syncProfileReference := 1;
   cmStackTableOutFrontAxisZ.commandConfiguration.camIn.masterStartDistance := 0.0;
   cmStackTableOutFrontAxisZ.commandConfiguration.camIn.velocity := -1.0;
   cmStackTableOutFrontAxisZ.commandConfiguration.camIn.acceleration := -1.0;
   cmStackTableOutFrontAxisZ.commandConfiguration.camIn.deceleration := -1.0;
   cmStackTableOutFrontAxisZ.commandConfiguration.camIn.jerk := -1.0;
   cmStackTableOutFrontAxisZ.commandConfiguration.camIn.applicationMode := 0;
   cmStackTableOutFrontAxisZ.commandConfiguration.camIn.syncDirection := 1;
   cmStackTableOutFrontAxisZ.commandConfiguration.gearOutCamOut.slavePosition := 0.0;
   cmStackTableOutFrontAxisZ.commandConfiguration.gearOutCamOut.syncProfileReference := 1;
   cmStackTableOutFrontAxisZ.commandConfiguration.gearOutCamOut.masterStopDistance := 0.0;
   cmStackTableOutFrontAxisZ.commandConfiguration.gearOutCamOut.deceleration := -1.0;
   cmStackTableOutFrontAxisZ.commandConfiguration.gearOutCamOut.jerk := -1.0;
   cmStackTableOutFrontAxisZ.commandConfiguration.gearOutCamOut.syncOutDirection := 3;
   cmStackTableOutFrontAxisZ.commandConfiguration.gearOutCamOut.gearOutCamOutMode := -1;
   cmStackTableOutFrontAxisZ.commandConfiguration.phasing.phaseShift := 0.0;
   cmStackTableOutFrontAxisZ.commandConfiguration.phasing.velocity := -1.0;
   cmStackTableOutFrontAxisZ.commandConfiguration.phasing.acceleration := -1.0;
   cmStackTableOutFrontAxisZ.commandConfiguration.phasing.deceleration := -1.0;
   cmStackTableOutFrontAxisZ.commandConfiguration.phasing.jerk := -1.0;
   cmStackTableOutFrontAxisZ.commandConfiguration.phasing.profileReference := 0;
   cmStackTableOutFrontAxisZ.commandConfiguration.phasing.phasingDistance := 0.0;
   cmStackTableOutFrontAxisZ.commandConfiguration.phasing.startPosition := 0.0;
   cmStackTableOutFrontAxisZ.commandConfiguration.phasing.direction := 3;
   cmStackTableOutFrontAxisZ.commandConfiguration.phasing.phaseAbsolute := TRUE;
   cmStackTableOutFrontAxisZ.commandConfiguration.phasing.phaseShiftChangeOnTheFly := FALSE;
   cmStackTableOutFrontAxisZ.commandConfiguration.offset.offset := 0.0;
   cmStackTableOutFrontAxisZ.commandConfiguration.offset.profileReference := 1;
   cmStackTableOutFrontAxisZ.commandConfiguration.offset.offsetDistance := 0.0;
   cmStackTableOutFrontAxisZ.commandConfiguration.offset.startPosition := 0.0;
   cmStackTableOutFrontAxisZ.commandConfiguration.offset.direction := 3;
   cmStackTableOutFrontAxisZ.commandConfiguration.offset.offsetAbsolute := TRUE;
   cmStackTableOutFrontAxisZ.commandConfiguration.offset.offsetChangeOnTheFly := FALSE;
   cmStackTableOutFrontAxisZ.commands.enableMasterControl := TRUE;
   cmStackTableOutFrontAxisZ.commands.enableAxis := FALSE;
   cmStackTableOutFrontAxisZ.commands.resetAxis := FALSE;
   cmStackTableOutFrontAxisZ.commands.openBrake := FALSE;
   cmStackTableOutFrontAxisZ.commands.jogForward := FALSE;
   cmStackTableOutFrontAxisZ.commands.jogBackward := FALSE;
   cmStackTableOutFrontAxisZ.commands.moveVelocity := FALSE;
   cmStackTableOutFrontAxisZ.commands.stop := FALSE;
   cmStackTableOutFrontAxisZ.commands.fastStop := FALSE;
   cmStackTableOutFrontAxisZ.commands.torqueLimiting := FALSE;
   cmStackTableOutFrontAxisZ.commands.homing := FALSE;
   cmStackTableOutFrontAxisZ.commands.posRelative := FALSE;
   cmStackTableOutFrontAxisZ.commands.posAbsolute := FALSE;
   cmStackTableOutFrontAxisZ.commands.posSuperimposed := FALSE;
   cmStackTableOutFrontAxisZ.commands.haltSuperimposed := FALSE;
   cmStackTableOutFrontAxisZ.commands.selectSetPosition := -1;
   cmStackTableOutFrontAxisZ.commands.uploadParameters := FALSE;
   cmStackTableOutFrontAxisZ.commands.refreshConfiguration := FALSE;
   cmStackTableOutFrontAxisZ.commands.editConfiguration := FALSE;
   cmStackTableOutFrontAxisZ.commands.saveConfiguration := FALSE;
   cmStackTableOutFrontAxisZ.commands.uploadCurrentTorque := FALSE;
   cmStackTableOutFrontAxisZ.commands.reset := FALSE;
   cmStackTableOutFrontAxisZ.monitoring.enable := TRUE;
   cmStackTableOutFrontAxisZ.monitoring.referenceDesignator := WSTRING#'StackTableOutFrontAxisZ';
   cmStackTableOutFrontAxisZ.monitoring.enabled := TRUE;
   cmStackTableOutFrontAxisZ.monitoring.enableManualCmds := FALSE;
   cmStackTableOutFrontAxisZ.monitoring.reset := FALSE;
   cmStackTableOutFrontAxisZ.monitoring.resetAxis := FALSE;
   cmStackTableOutFrontAxisZ.monitoring.enableAxis := TRUE;
   cmStackTableOutFrontAxisZ.monitoring.openBrake := FALSE;
   cmStackTableOutFrontAxisZ.monitoring.jogBackward := FALSE;
   cmStackTableOutFrontAxisZ.monitoring.jogForward := FALSE;
   cmStackTableOutFrontAxisZ.monitoring.moveVelocity := FALSE;
   cmStackTableOutFrontAxisZ.monitoring.stop := FALSE;
   cmStackTableOutFrontAxisZ.monitoring.fastStop := FALSE;
   cmStackTableOutFrontAxisZ.monitoring.torqueLimiting := FALSE;
   cmStackTableOutFrontAxisZ.monitoring.homing := FALSE;
   cmStackTableOutFrontAxisZ.monitoring.posRelative := FALSE;
   cmStackTableOutFrontAxisZ.monitoring.posAbsolute := FALSE;
   cmStackTableOutFrontAxisZ.monitoring.posSuperimposed := FALSE;
   cmStackTableOutFrontAxisZ.monitoring.haltSuperimposed := FALSE;
   cmStackTableOutFrontAxisZ.monitoring.brakeOpened := FALSE;
   cmStackTableOutFrontAxisZ.monitoring.axisEnabled := TRUE;
   cmStackTableOutFrontAxisZ.monitoring.resetActive := FALSE;
   cmStackTableOutFrontAxisZ.monitoring.inVelocity := FALSE;
   cmStackTableOutFrontAxisZ.monitoring.inLimitation := FALSE;
   cmStackTableOutFrontAxisZ.monitoring.inClamping := FALSE;
   cmStackTableOutFrontAxisZ.monitoring.startSync := FALSE;
   cmStackTableOutFrontAxisZ.monitoring.inSync := FALSE;
   cmStackTableOutFrontAxisZ.monitoring.inSimulation := FALSE;
   cmStackTableOutFrontAxisZ.monitoring.jogSelected := FALSE;
   cmStackTableOutFrontAxisZ.monitoring.moveVelocitySelected := FALSE;
   cmStackTableOutFrontAxisZ.monitoring.stopSelected := FALSE;
   cmStackTableOutFrontAxisZ.monitoring.fastStopSelected := FALSE;
   cmStackTableOutFrontAxisZ.monitoring.torqueLimitingSelected := FALSE;
   cmStackTableOutFrontAxisZ.monitoring.homingSelected := FALSE;
   cmStackTableOutFrontAxisZ.monitoring.posRelativeSelected := FALSE;
   cmStackTableOutFrontAxisZ.monitoring.posAbsoluteSelected := FALSE;
   cmStackTableOutFrontAxisZ.monitoring.posSuperimposedSelected := FALSE;
   cmStackTableOutFrontAxisZ.monitoring.haltSuperimposedSelected := FALSE;
   cmStackTableOutFrontAxisZ.monitoring.commandBusy := FALSE;
   cmStackTableOutFrontAxisZ.monitoring.commandDone := FALSE;
   cmStackTableOutFrontAxisZ.monitoring.commandAborted := FALSE;
   cmStackTableOutFrontAxisZ.monitoring.homingCommandBusy := FALSE;
   cmStackTableOutFrontAxisZ.monitoring.homingCommandDone := FALSE;
   cmStackTableOutFrontAxisZ.monitoring.homingCommandAborted := FALSE;
   cmStackTableOutFrontAxisZ.monitoring.superimposedBusy := FALSE;
   cmStackTableOutFrontAxisZ.monitoring.superimposedDone := FALSE;
   cmStackTableOutFrontAxisZ.monitoring.superimposedAborted := FALSE;
   cmStackTableOutFrontAxisZ.monitoring.selectSetPosition := -1;
   cmStackTableOutFrontAxisZ.monitoring.selectionController := FALSE;
   cmStackTableOutFrontAxisZ.monitoring.interlockGeneral := TRUE;
   cmStackTableOutFrontAxisZ.monitoring.interlockJogForward := TRUE;
   cmStackTableOutFrontAxisZ.monitoring.interlockJogBackward := TRUE;
   cmStackTableOutFrontAxisZ.monitoring.interlockWarningGeneral := FALSE;
   cmStackTableOutFrontAxisZ.monitoring.interlockWarningJogForward := FALSE;
   cmStackTableOutFrontAxisZ.monitoring.interlockWarningJogBackward := FALSE;
   cmStackTableOutFrontAxisZ.monitoring.valid := TRUE;
   cmStackTableOutFrontAxisZ.monitoring.busy := TRUE;
   cmStackTableOutFrontAxisZ.monitoring.error := FALSE;
   cmStackTableOutFrontAxisZ.monitoring.status := 16#7002;
   cmStackTableOutFrontAxisZ.monitoring.subfunctionStatus := 16#0000;
   cmStackTableOutFrontAxisZ.monitoring.actualPosition := 0.0;
   cmStackTableOutFrontAxisZ.monitoring.actualSpeed := 0.0;
   cmStackTableOutFrontAxisZ.monitoring.speedUnit := 1062;
   cmStackTableOutFrontAxisZ.monitoring.positionUnit := 1013;
   cmStackTableOutFrontAxisZ.monitoring.axisStatus1 := 16#0200_10E1;
   cmStackTableOutFrontAxisZ.monitoring.axisStatus2 := 16#0000_0000;
   cmStackTableOutFrontAxisZ.monitoring.axisType := 1;
   cmStackTableOutFrontAxisZ.monitoring.maxVelocity := 2500.0;
   cmStackTableOutFrontAxisZ.monitoring.actualCurrent := 0.0;
   cmStackTableOutFrontAxisZ.monitoring.actualTorque := 0.0;
   cmStackTableOutFrontAxisZ.monitoring.velocityOverrideEnabled := FALSE;
   cmStackTableOutFrontAxisZ.monitoring.sinaParaError := FALSE;
   cmStackTableOutFrontAxisZ.monitoring.sinaParaStatus := 16#0000_0000;
   cmStackTableOutFrontAxisZ.configuration.referenceDesignator := WSTRING#'StackTableOutFrontAxisZ';
   cmStackTableOutFrontAxisZ.configuration.disableAlarms := FALSE;
   cmStackTableOutFrontAxisZ.configuration.masterControlPopUp := TRUE;
   cmStackTableOutFrontAxisZ.configuration.setPositions[0].position := 0.0;
   cmStackTableOutFrontAxisZ.configuration.setPositions[1].position := 500.0;
   cmStackTableOutFrontAxisZ.configuration.setPositions[2..15].position := 0.0;
   cmStackTableOutFrontAxisZ.configuration.setPositions[0..1].velocity := 500.0;
   cmStackTableOutFrontAxisZ.configuration.setPositions[2..15].velocity := -1.0;
   cmStackTableOutFrontAxisZ.configuration.setPositions[0..1].acceleration := 5000.0;
   cmStackTableOutFrontAxisZ.configuration.setPositions[2..15].acceleration := -1.0;
   cmStackTableOutFrontAxisZ.configuration.setPositions[0..1].deceleration := 5000.0;
   cmStackTableOutFrontAxisZ.configuration.setPositions[2..15].deceleration := -1.0;
   cmStackTableOutFrontAxisZ.configuration.setPositions[0..15]."name" := '';
   cmStackTableOutRearAxisZ.commandConfiguration.generalSettings.stopOnError := TRUE;
   cmStackTableOutRearAxisZ.commandConfiguration.generalSettings.resetWithRestart := FALSE;
   cmStackTableOutRearAxisZ.commandConfiguration.generalSettings.abortWaitingSyncCmd := TRUE;
   cmStackTableOutRearAxisZ.commandConfiguration.power.startMode := 1;
   cmStackTableOutRearAxisZ.commandConfiguration.power.stopMode := 0;
   cmStackTableOutRearAxisZ.commandConfiguration.power.syncMotionSimulation := FALSE;
   cmStackTableOutRearAxisZ.commandConfiguration.power.syncMotionSimulationExtendedMode := -1;
   cmStackTableOutRearAxisZ.commandConfiguration.jog.velocity := 0.0;
   cmStackTableOutRearAxisZ.commandConfiguration.jog.acceleration := -1.0;
   cmStackTableOutRearAxisZ.commandConfiguration.jog.deceleration := -1.0;
   cmStackTableOutRearAxisZ.commandConfiguration.jog.jerk := -1.0;
   cmStackTableOutRearAxisZ.commandConfiguration.jog.positionControlled := TRUE;
   cmStackTableOutRearAxisZ.commandConfiguration.jog.increment := 0.0;
   cmStackTableOutRearAxisZ.commandConfiguration.jog.mode := 0;
   cmStackTableOutRearAxisZ.commandConfiguration.moveVelocity.velocity := 0.0;
   cmStackTableOutRearAxisZ.commandConfiguration.moveVelocity.acceleration := -1.0;
   cmStackTableOutRearAxisZ.commandConfiguration.moveVelocity.deceleration := -1.0;
   cmStackTableOutRearAxisZ.commandConfiguration.moveVelocity.jerk := -1.0;
   cmStackTableOutRearAxisZ.commandConfiguration.moveVelocity.direction := 0;
   cmStackTableOutRearAxisZ.commandConfiguration.moveVelocity.positionControlled := TRUE;
   cmStackTableOutRearAxisZ.commandConfiguration.moveVelocity.velocityChangeOnTheFly := FALSE;
   cmStackTableOutRearAxisZ.commandConfiguration.stop.deceleration := -1.0;
   cmStackTableOutRearAxisZ.commandConfiguration.stop.jerk := -1.0;
   cmStackTableOutRearAxisZ.commandConfiguration.stop.abortAcceleration := FALSE;
   cmStackTableOutRearAxisZ.commandConfiguration.fastStop.deceleration := -1.0;
   cmStackTableOutRearAxisZ.commandConfiguration.fastStop.jerk := -1.0;
   cmStackTableOutRearAxisZ.commandConfiguration.fastStop.abortAcceleration := FALSE;
   cmStackTableOutRearAxisZ.commandConfiguration.fastStop.replaceStopPossible := FALSE;
   cmStackTableOutRearAxisZ.commandConfiguration.torqueLimiting.limit := -1.0;
   cmStackTableOutRearAxisZ.commandConfiguration.torqueLimiting.mode := 0;
   cmStackTableOutRearAxisZ.commandConfiguration.homing.position := 0.0;
   cmStackTableOutRearAxisZ.commandConfiguration.homing.mode := 0;
   cmStackTableOutRearAxisZ.commandConfiguration.homing.sensor := 0;
   cmStackTableOutRearAxisZ.commandConfiguration.homing.extendedMode := -1;
   cmStackTableOutRearAxisZ.commandConfiguration.homing.extendedModeTorqueLimit := 0.0;
   cmStackTableOutRearAxisZ.commandConfiguration.homing.extendedModeTargetPosition := 0.0;
   cmStackTableOutRearAxisZ.commandConfiguration.posRelative.distance := 0.0;
   cmStackTableOutRearAxisZ.commandConfiguration.posRelative.velocity := -1.0;
   cmStackTableOutRearAxisZ.commandConfiguration.posRelative.acceleration := -1.0;
   cmStackTableOutRearAxisZ.commandConfiguration.posRelative.deceleration := -1.0;
   cmStackTableOutRearAxisZ.commandConfiguration.posRelative.jerk := -1.0;
   cmStackTableOutRearAxisZ.commandConfiguration.posRelative.direction := 0;
   cmStackTableOutRearAxisZ.commandConfiguration.posAbsolute.position := 0.0;
   cmStackTableOutRearAxisZ.commandConfiguration.posAbsolute.velocity := -1.0;
   cmStackTableOutRearAxisZ.commandConfiguration.posAbsolute.acceleration := -1.0;
   cmStackTableOutRearAxisZ.commandConfiguration.posAbsolute.deceleration := -1.0;
   cmStackTableOutRearAxisZ.commandConfiguration.posAbsolute.jerk := -1.0;
   cmStackTableOutRearAxisZ.commandConfiguration.posAbsolute.direction := 1;
   cmStackTableOutRearAxisZ.commandConfiguration.posAbsolute.positionChangeOnTheFly := FALSE;
   cmStackTableOutRearAxisZ.commandConfiguration.posAbsolute.velocityChangeOnTheFly := FALSE;
   cmStackTableOutRearAxisZ.commandConfiguration.posSuperimposed.distance := 0.0;
   cmStackTableOutRearAxisZ.commandConfiguration.posSuperimposed.velocityDiff := -1.0;
   cmStackTableOutRearAxisZ.commandConfiguration.posSuperimposed.acceleration := -1.0;
   cmStackTableOutRearAxisZ.commandConfiguration.posSuperimposed.deceleration := -1.0;
   cmStackTableOutRearAxisZ.commandConfiguration.posSuperimposed.jerk := -1.0;
   cmStackTableOutRearAxisZ.commandConfiguration.posSuperimposed.direction := 0;
   cmStackTableOutRearAxisZ.commandConfiguration.haltSuperimposed.deceleration := -1.0;
   cmStackTableOutRearAxisZ.commandConfiguration.haltSuperimposed.jerk := -1.0;
   cmStackTableOutRearAxisZ.commandConfiguration.haltSuperimposed.abortAcceleration := FALSE;
   cmStackTableOutRearAxisZ.commandConfiguration.gearInRelative.ratioNumerator := 1;
   cmStackTableOutRearAxisZ.commandConfiguration.gearInRelative.ratioDenominator := 1;
   cmStackTableOutRearAxisZ.commandConfiguration.gearInRelative.acceleration := -1.0;
   cmStackTableOutRearAxisZ.commandConfiguration.gearInRelative.deceleration := -1.0;
   cmStackTableOutRearAxisZ.commandConfiguration.gearInRelative.jerk := -1.0;
   cmStackTableOutRearAxisZ.commandConfiguration.gearInRelative.ratioChangeOnTheFly := FALSE;
   cmStackTableOutRearAxisZ.commandConfiguration.gearInAbsolute.ratioNumerator := 1;
   cmStackTableOutRearAxisZ.commandConfiguration.gearInAbsolute.ratioDenominator := 1;
   cmStackTableOutRearAxisZ.commandConfiguration.gearInAbsolute.masterSyncPosition := 0.0;
   cmStackTableOutRearAxisZ.commandConfiguration.gearInAbsolute.slaveSyncPosition := 0.0;
   cmStackTableOutRearAxisZ.commandConfiguration.gearInAbsolute.syncProfileReference := 1;
   cmStackTableOutRearAxisZ.commandConfiguration.gearInAbsolute.masterStartDistance := 0.0;
   cmStackTableOutRearAxisZ.commandConfiguration.gearInAbsolute.velocity := -1.0;
   cmStackTableOutRearAxisZ.commandConfiguration.gearInAbsolute.acceleration := -1.0;
   cmStackTableOutRearAxisZ.commandConfiguration.gearInAbsolute.deceleration := -1.0;
   cmStackTableOutRearAxisZ.commandConfiguration.gearInAbsolute.jerk := -1.0;
   cmStackTableOutRearAxisZ.commandConfiguration.gearInAbsolute.syncDirection := 1;
   cmStackTableOutRearAxisZ.commandConfiguration.gearInAbsolute.ratioChangeOnTheFly := FALSE;
   cmStackTableOutRearAxisZ.commandConfiguration.gearInVelocity.continuousUpdate := FALSE;
   cmStackTableOutRearAxisZ.commandConfiguration.gearInVelocity.ratioNumerator := 1;
   cmStackTableOutRearAxisZ.commandConfiguration.gearInVelocity.ratioDenominator := 1;
   cmStackTableOutRearAxisZ.commandConfiguration.gearInVelocity.acceleration := -1.0;
   cmStackTableOutRearAxisZ.commandConfiguration.gearInVelocity.deceleration := -1.0;
   cmStackTableOutRearAxisZ.commandConfiguration.gearInVelocity.jerk := -1.0;
   cmStackTableOutRearAxisZ.commandConfiguration.gearInVelocity.positionControlled := FALSE;
   cmStackTableOutRearAxisZ.commandConfiguration.camIn.masterOffset := 0.0;
   cmStackTableOutRearAxisZ.commandConfiguration.camIn.slaveOffset := 0.0;
   cmStackTableOutRearAxisZ.commandConfiguration.camIn.masterScaling := 1.0;
   cmStackTableOutRearAxisZ.commandConfiguration.camIn.slaveScaling := 1.0;
   cmStackTableOutRearAxisZ.commandConfiguration.camIn.masterSyncPosition := 0.0;
   cmStackTableOutRearAxisZ.commandConfiguration.camIn.syncProfileReference := 1;
   cmStackTableOutRearAxisZ.commandConfiguration.camIn.masterStartDistance := 0.0;
   cmStackTableOutRearAxisZ.commandConfiguration.camIn.velocity := -1.0;
   cmStackTableOutRearAxisZ.commandConfiguration.camIn.acceleration := -1.0;
   cmStackTableOutRearAxisZ.commandConfiguration.camIn.deceleration := -1.0;
   cmStackTableOutRearAxisZ.commandConfiguration.camIn.jerk := -1.0;
   cmStackTableOutRearAxisZ.commandConfiguration.camIn.applicationMode := 0;
   cmStackTableOutRearAxisZ.commandConfiguration.camIn.syncDirection := 1;
   cmStackTableOutRearAxisZ.commandConfiguration.gearOutCamOut.slavePosition := 0.0;
   cmStackTableOutRearAxisZ.commandConfiguration.gearOutCamOut.syncProfileReference := 1;
   cmStackTableOutRearAxisZ.commandConfiguration.gearOutCamOut.masterStopDistance := 0.0;
   cmStackTableOutRearAxisZ.commandConfiguration.gearOutCamOut.deceleration := -1.0;
   cmStackTableOutRearAxisZ.commandConfiguration.gearOutCamOut.jerk := -1.0;
   cmStackTableOutRearAxisZ.commandConfiguration.gearOutCamOut.syncOutDirection := 3;
   cmStackTableOutRearAxisZ.commandConfiguration.gearOutCamOut.gearOutCamOutMode := -1;
   cmStackTableOutRearAxisZ.commandConfiguration.phasing.phaseShift := 0.0;
   cmStackTableOutRearAxisZ.commandConfiguration.phasing.velocity := -1.0;
   cmStackTableOutRearAxisZ.commandConfiguration.phasing.acceleration := -1.0;
   cmStackTableOutRearAxisZ.commandConfiguration.phasing.deceleration := -1.0;
   cmStackTableOutRearAxisZ.commandConfiguration.phasing.jerk := -1.0;
   cmStackTableOutRearAxisZ.commandConfiguration.phasing.profileReference := 0;
   cmStackTableOutRearAxisZ.commandConfiguration.phasing.phasingDistance := 0.0;
   cmStackTableOutRearAxisZ.commandConfiguration.phasing.startPosition := 0.0;
   cmStackTableOutRearAxisZ.commandConfiguration.phasing.direction := 3;
   cmStackTableOutRearAxisZ.commandConfiguration.phasing.phaseAbsolute := TRUE;
   cmStackTableOutRearAxisZ.commandConfiguration.phasing.phaseShiftChangeOnTheFly := FALSE;
   cmStackTableOutRearAxisZ.commandConfiguration.offset.offset := 0.0;
   cmStackTableOutRearAxisZ.commandConfiguration.offset.profileReference := 1;
   cmStackTableOutRearAxisZ.commandConfiguration.offset.offsetDistance := 0.0;
   cmStackTableOutRearAxisZ.commandConfiguration.offset.startPosition := 0.0;
   cmStackTableOutRearAxisZ.commandConfiguration.offset.direction := 3;
   cmStackTableOutRearAxisZ.commandConfiguration.offset.offsetAbsolute := TRUE;
   cmStackTableOutRearAxisZ.commandConfiguration.offset.offsetChangeOnTheFly := FALSE;
   cmStackTableOutRearAxisZ.commands.enableMasterControl := TRUE;
   cmStackTableOutRearAxisZ.commands.enableAxis := FALSE;
   cmStackTableOutRearAxisZ.commands.resetAxis := FALSE;
   cmStackTableOutRearAxisZ.commands.openBrake := FALSE;
   cmStackTableOutRearAxisZ.commands.jogForward := FALSE;
   cmStackTableOutRearAxisZ.commands.jogBackward := FALSE;
   cmStackTableOutRearAxisZ.commands.moveVelocity := FALSE;
   cmStackTableOutRearAxisZ.commands.stop := FALSE;
   cmStackTableOutRearAxisZ.commands.fastStop := FALSE;
   cmStackTableOutRearAxisZ.commands.torqueLimiting := FALSE;
   cmStackTableOutRearAxisZ.commands.homing := FALSE;
   cmStackTableOutRearAxisZ.commands.posRelative := FALSE;
   cmStackTableOutRearAxisZ.commands.posAbsolute := FALSE;
   cmStackTableOutRearAxisZ.commands.posSuperimposed := FALSE;
   cmStackTableOutRearAxisZ.commands.haltSuperimposed := FALSE;
   cmStackTableOutRearAxisZ.commands.selectSetPosition := -1;
   cmStackTableOutRearAxisZ.commands.uploadParameters := FALSE;
   cmStackTableOutRearAxisZ.commands.refreshConfiguration := FALSE;
   cmStackTableOutRearAxisZ.commands.editConfiguration := FALSE;
   cmStackTableOutRearAxisZ.commands.saveConfiguration := FALSE;
   cmStackTableOutRearAxisZ.commands.uploadCurrentTorque := FALSE;
   cmStackTableOutRearAxisZ.commands.reset := FALSE;
   cmStackTableOutRearAxisZ.monitoring.enable := TRUE;
   cmStackTableOutRearAxisZ.monitoring.referenceDesignator := WSTRING#'StackTableOutRearAxisZ';
   cmStackTableOutRearAxisZ.monitoring.enabled := TRUE;
   cmStackTableOutRearAxisZ.monitoring.enableManualCmds := FALSE;
   cmStackTableOutRearAxisZ.monitoring.reset := FALSE;
   cmStackTableOutRearAxisZ.monitoring.resetAxis := FALSE;
   cmStackTableOutRearAxisZ.monitoring.enableAxis := TRUE;
   cmStackTableOutRearAxisZ.monitoring.openBrake := FALSE;
   cmStackTableOutRearAxisZ.monitoring.jogBackward := FALSE;
   cmStackTableOutRearAxisZ.monitoring.jogForward := FALSE;
   cmStackTableOutRearAxisZ.monitoring.moveVelocity := FALSE;
   cmStackTableOutRearAxisZ.monitoring.stop := FALSE;
   cmStackTableOutRearAxisZ.monitoring.fastStop := FALSE;
   cmStackTableOutRearAxisZ.monitoring.torqueLimiting := FALSE;
   cmStackTableOutRearAxisZ.monitoring.homing := FALSE;
   cmStackTableOutRearAxisZ.monitoring.posRelative := FALSE;
   cmStackTableOutRearAxisZ.monitoring.posAbsolute := FALSE;
   cmStackTableOutRearAxisZ.monitoring.posSuperimposed := FALSE;
   cmStackTableOutRearAxisZ.monitoring.haltSuperimposed := FALSE;
   cmStackTableOutRearAxisZ.monitoring.brakeOpened := FALSE;
   cmStackTableOutRearAxisZ.monitoring.axisEnabled := TRUE;
   cmStackTableOutRearAxisZ.monitoring.resetActive := FALSE;
   cmStackTableOutRearAxisZ.monitoring.inVelocity := FALSE;
   cmStackTableOutRearAxisZ.monitoring.inLimitation := FALSE;
   cmStackTableOutRearAxisZ.monitoring.inClamping := FALSE;
   cmStackTableOutRearAxisZ.monitoring.startSync := FALSE;
   cmStackTableOutRearAxisZ.monitoring.inSync := FALSE;
   cmStackTableOutRearAxisZ.monitoring.inSimulation := FALSE;
   cmStackTableOutRearAxisZ.monitoring.jogSelected := FALSE;
   cmStackTableOutRearAxisZ.monitoring.moveVelocitySelected := FALSE;
   cmStackTableOutRearAxisZ.monitoring.stopSelected := FALSE;
   cmStackTableOutRearAxisZ.monitoring.fastStopSelected := FALSE;
   cmStackTableOutRearAxisZ.monitoring.torqueLimitingSelected := FALSE;
   cmStackTableOutRearAxisZ.monitoring.homingSelected := FALSE;
   cmStackTableOutRearAxisZ.monitoring.posRelativeSelected := FALSE;
   cmStackTableOutRearAxisZ.monitoring.posAbsoluteSelected := FALSE;
   cmStackTableOutRearAxisZ.monitoring.posSuperimposedSelected := FALSE;
   cmStackTableOutRearAxisZ.monitoring.haltSuperimposedSelected := FALSE;
   cmStackTableOutRearAxisZ.monitoring.commandBusy := FALSE;
   cmStackTableOutRearAxisZ.monitoring.commandDone := FALSE;
   cmStackTableOutRearAxisZ.monitoring.commandAborted := FALSE;
   cmStackTableOutRearAxisZ.monitoring.homingCommandBusy := FALSE;
   cmStackTableOutRearAxisZ.monitoring.homingCommandDone := FALSE;
   cmStackTableOutRearAxisZ.monitoring.homingCommandAborted := FALSE;
   cmStackTableOutRearAxisZ.monitoring.superimposedBusy := FALSE;
   cmStackTableOutRearAxisZ.monitoring.superimposedDone := FALSE;
   cmStackTableOutRearAxisZ.monitoring.superimposedAborted := FALSE;
   cmStackTableOutRearAxisZ.monitoring.selectSetPosition := -1;
   cmStackTableOutRearAxisZ.monitoring.selectionController := FALSE;
   cmStackTableOutRearAxisZ.monitoring.interlockGeneral := TRUE;
   cmStackTableOutRearAxisZ.monitoring.interlockJogForward := TRUE;
   cmStackTableOutRearAxisZ.monitoring.interlockJogBackward := TRUE;
   cmStackTableOutRearAxisZ.monitoring.interlockWarningGeneral := FALSE;
   cmStackTableOutRearAxisZ.monitoring.interlockWarningJogForward := FALSE;
   cmStackTableOutRearAxisZ.monitoring.interlockWarningJogBackward := FALSE;
   cmStackTableOutRearAxisZ.monitoring.valid := TRUE;
   cmStackTableOutRearAxisZ.monitoring.busy := TRUE;
   cmStackTableOutRearAxisZ.monitoring.error := FALSE;
   cmStackTableOutRearAxisZ.monitoring.status := 16#7002;
   cmStackTableOutRearAxisZ.monitoring.subfunctionStatus := 16#0000;
   cmStackTableOutRearAxisZ.monitoring.actualPosition := 0.0;
   cmStackTableOutRearAxisZ.monitoring.actualSpeed := 0.0;
   cmStackTableOutRearAxisZ.monitoring.speedUnit := 1062;
   cmStackTableOutRearAxisZ.monitoring.positionUnit := 1013;
   cmStackTableOutRearAxisZ.monitoring.axisStatus1 := 16#0200_10E1;
   cmStackTableOutRearAxisZ.monitoring.axisStatus2 := 16#0000_0000;
   cmStackTableOutRearAxisZ.monitoring.axisType := 1;
   cmStackTableOutRearAxisZ.monitoring.maxVelocity := 2500.0;
   cmStackTableOutRearAxisZ.monitoring.actualCurrent := 0.0;
   cmStackTableOutRearAxisZ.monitoring.actualTorque := 0.0;
   cmStackTableOutRearAxisZ.monitoring.velocityOverrideEnabled := FALSE;
   cmStackTableOutRearAxisZ.monitoring.sinaParaError := FALSE;
   cmStackTableOutRearAxisZ.monitoring.sinaParaStatus := 16#0000_0000;
   cmStackTableOutRearAxisZ.configuration.referenceDesignator := WSTRING#'StackTableOutRearAxisZ';
   cmStackTableOutRearAxisZ.configuration.disableAlarms := FALSE;
   cmStackTableOutRearAxisZ.configuration.masterControlPopUp := TRUE;
   cmStackTableOutRearAxisZ.configuration.setPositions[0].position := 0.0;
   cmStackTableOutRearAxisZ.configuration.setPositions[1].position := 500.0;
   cmStackTableOutRearAxisZ.configuration.setPositions[2..15].position := 0.0;
   cmStackTableOutRearAxisZ.configuration.setPositions[0..1].velocity := 500.0;
   cmStackTableOutRearAxisZ.configuration.setPositions[2..15].velocity := -1.0;
   cmStackTableOutRearAxisZ.configuration.setPositions[0..1].acceleration := 5000.0;
   cmStackTableOutRearAxisZ.configuration.setPositions[2..15].acceleration := -1.0;
   cmStackTableOutRearAxisZ.configuration.setPositions[0..1].deceleration := 5000.0;
   cmStackTableOutRearAxisZ.configuration.setPositions[2..15].deceleration := -1.0;
   cmStackTableOutRearAxisZ.configuration.setPositions[0..15]."name" := '';
   cmMendrelAnodeFrontClamp.commands.refreshConfiguration := FALSE;
   cmMendrelAnodeFrontClamp.commands.editConfiguration := FALSE;
   cmMendrelAnodeFrontClamp.commands.saveConfiguration := FALSE;
   cmMendrelAnodeFrontClamp.commands.reset := FALSE;
   cmMendrelAnodeFrontClamp.commands.commandHomePos := FALSE;
   cmMendrelAnodeFrontClamp.commands.commandWorkPos := FALSE;
   cmMendrelAnodeFrontClamp.monitoring.enable := TRUE;
   cmMendrelAnodeFrontClamp.monitoring.referenceDesignator := WSTRING#'MendrelAnodeFrontClamp';
   cmMendrelAnodeFrontClamp.monitoring.commandHomePos := FALSE;
   cmMendrelAnodeFrontClamp.monitoring.commandWorkPos := FALSE;
   cmMendrelAnodeFrontClamp.monitoring.goToHomePos := FALSE;
   cmMendrelAnodeFrontClamp.monitoring.goToWorkPos := TRUE;
   cmMendrelAnodeFrontClamp.monitoring.inHomePos := FALSE;
   cmMendrelAnodeFrontClamp.monitoring.inWorkPos := TRUE;
   cmMendrelAnodeFrontClamp.monitoring.reset := FALSE;
   cmMendrelAnodeFrontClamp.monitoring.enableManualCmds := FALSE;
   cmMendrelAnodeFrontClamp.monitoring.error := FALSE;
   cmMendrelAnodeFrontClamp.monitoring.interlockHomePos := TRUE;
   cmMendrelAnodeFrontClamp.monitoring.interlockWorkPos := TRUE;
   cmMendrelAnodeFrontClamp.monitoring.status := 16#7006;
   cmMendrelAnodeFrontClamp.monitoring.interlockWarningWorkPos := FALSE;
   cmMendrelAnodeFrontClamp.monitoring.interlockWarningHomePos := FALSE;
   cmMendrelAnodeFrontClamp.configuration.referenceDesignator := WSTRING#'TwoWayAct.';
   cmMendrelAnodeFrontClamp.configuration.monitoringLeavingFeedback := T#5S;
   cmMendrelAnodeFrontClamp.configuration.monitoringReachingFeedback := T#5S;
   cmMendrelAnodeFrontClamp.configuration.monitoringDiscrepancy := T#0MS;
   cmMendrelAnodeFrontClamp.configuration.setOutputHomeContinuously := TRUE;
   cmMendrelAnodeFrontClamp.configuration.setOutputWorkContinuously := TRUE;
   cmMendrelAnodeFrontClamp.configuration.disableHomeCommand := FALSE;
   cmMendrelAnodeFrontClamp.configuration.disableFeedbackHomePos := FALSE;
   cmMendrelAnodeFrontClamp.configuration.disableFeedbackWorkPos := FALSE;
   cmMendrelAnodeFrontClamp.configuration.disableAlarms := FALSE;
   cmMendrelAnodeFrontClamp.configuration.resetOutputsOnError := FALSE;
   cmMendrelAnodeFrontClamp.configuration.allwaysWaitOnReachingTime := FALSE;
   cmMendrelAnodeRearClamp.commands.refreshConfiguration := FALSE;
   cmMendrelAnodeRearClamp.commands.editConfiguration := FALSE;
   cmMendrelAnodeRearClamp.commands.saveConfiguration := FALSE;
   cmMendrelAnodeRearClamp.commands.reset := FALSE;
   cmMendrelAnodeRearClamp.commands.commandHomePos := FALSE;
   cmMendrelAnodeRearClamp.commands.commandWorkPos := FALSE;
   cmMendrelAnodeRearClamp.monitoring.enable := TRUE;
   cmMendrelAnodeRearClamp.monitoring.referenceDesignator := WSTRING#'MendrelAnodeRearClamp';
   cmMendrelAnodeRearClamp.monitoring.commandHomePos := FALSE;
   cmMendrelAnodeRearClamp.monitoring.commandWorkPos := FALSE;
   cmMendrelAnodeRearClamp.monitoring.goToHomePos := FALSE;
   cmMendrelAnodeRearClamp.monitoring.goToWorkPos := TRUE;
   cmMendrelAnodeRearClamp.monitoring.inHomePos := FALSE;
   cmMendrelAnodeRearClamp.monitoring.inWorkPos := TRUE;
   cmMendrelAnodeRearClamp.monitoring.reset := FALSE;
   cmMendrelAnodeRearClamp.monitoring.enableManualCmds := FALSE;
   cmMendrelAnodeRearClamp.monitoring.error := FALSE;
   cmMendrelAnodeRearClamp.monitoring.interlockHomePos := TRUE;
   cmMendrelAnodeRearClamp.monitoring.interlockWorkPos := TRUE;
   cmMendrelAnodeRearClamp.monitoring.status := 16#7006;
   cmMendrelAnodeRearClamp.monitoring.interlockWarningWorkPos := FALSE;
   cmMendrelAnodeRearClamp.monitoring.interlockWarningHomePos := FALSE;
   cmMendrelAnodeRearClamp.configuration.referenceDesignator := WSTRING#'TwoWayAct.';
   cmMendrelAnodeRearClamp.configuration.monitoringLeavingFeedback := T#5S;
   cmMendrelAnodeRearClamp.configuration.monitoringReachingFeedback := T#5S;
   cmMendrelAnodeRearClamp.configuration.monitoringDiscrepancy := T#0MS;
   cmMendrelAnodeRearClamp.configuration.setOutputHomeContinuously := TRUE;
   cmMendrelAnodeRearClamp.configuration.setOutputWorkContinuously := TRUE;
   cmMendrelAnodeRearClamp.configuration.disableHomeCommand := FALSE;
   cmMendrelAnodeRearClamp.configuration.disableFeedbackHomePos := FALSE;
   cmMendrelAnodeRearClamp.configuration.disableFeedbackWorkPos := FALSE;
   cmMendrelAnodeRearClamp.configuration.disableAlarms := FALSE;
   cmMendrelAnodeRearClamp.configuration.resetOutputsOnError := FALSE;
   cmMendrelAnodeRearClamp.configuration.allwaysWaitOnReachingTime := FALSE;
   cmMendrelCathodeFrontClamp.commands.refreshConfiguration := FALSE;
   cmMendrelCathodeFrontClamp.commands.editConfiguration := FALSE;
   cmMendrelCathodeFrontClamp.commands.saveConfiguration := FALSE;
   cmMendrelCathodeFrontClamp.commands.reset := FALSE;
   cmMendrelCathodeFrontClamp.commands.commandHomePos := FALSE;
   cmMendrelCathodeFrontClamp.commands.commandWorkPos := FALSE;
   cmMendrelCathodeFrontClamp.monitoring.enable := TRUE;
   cmMendrelCathodeFrontClamp.monitoring.referenceDesignator := WSTRING#'MendrelCathodeFrontClamp';
   cmMendrelCathodeFrontClamp.monitoring.commandHomePos := FALSE;
   cmMendrelCathodeFrontClamp.monitoring.commandWorkPos := FALSE;
   cmMendrelCathodeFrontClamp.monitoring.goToHomePos := FALSE;
   cmMendrelCathodeFrontClamp.monitoring.goToWorkPos := TRUE;
   cmMendrelCathodeFrontClamp.monitoring.inHomePos := FALSE;
   cmMendrelCathodeFrontClamp.monitoring.inWorkPos := TRUE;
   cmMendrelCathodeFrontClamp.monitoring.reset := FALSE;
   cmMendrelCathodeFrontClamp.monitoring.enableManualCmds := FALSE;
   cmMendrelCathodeFrontClamp.monitoring.error := FALSE;
   cmMendrelCathodeFrontClamp.monitoring.interlockHomePos := TRUE;
   cmMendrelCathodeFrontClamp.monitoring.interlockWorkPos := TRUE;
   cmMendrelCathodeFrontClamp.monitoring.status := 16#7006;
   cmMendrelCathodeFrontClamp.monitoring.interlockWarningWorkPos := FALSE;
   cmMendrelCathodeFrontClamp.monitoring.interlockWarningHomePos := FALSE;
   cmMendrelCathodeFrontClamp.configuration.referenceDesignator := WSTRING#'TwoWayAct.';
   cmMendrelCathodeFrontClamp.configuration.monitoringLeavingFeedback := T#5S;
   cmMendrelCathodeFrontClamp.configuration.monitoringReachingFeedback := T#5S;
   cmMendrelCathodeFrontClamp.configuration.monitoringDiscrepancy := T#0MS;
   cmMendrelCathodeFrontClamp.configuration.setOutputHomeContinuously := TRUE;
   cmMendrelCathodeFrontClamp.configuration.setOutputWorkContinuously := TRUE;
   cmMendrelCathodeFrontClamp.configuration.disableHomeCommand := FALSE;
